LIN {X 0,Y 399.766,Z 653.208,A -85,B 0,C 180,E1 19416.646,E2 19416.646} C_VEL
LIN {X 0,Y 400.216,Z 637.351,A -85,B 0,C 180,E1 19415.617,E2 19415.617} C_VEL
LIN {X 0,Y 400.424,Z 621.306,A -85,B 0,C 180,E1 19414.872,E2 19414.872} C_VEL
LIN {X 0,Y 400.403,Z 603.741,A -85,B 0,C 180,E1 19414.34,E2 19414.34} C_VEL
LIN {X 0,Y 401.742,Z 547.411,A -85,B 0,C 180,E1 19413.015,E2 19413.015} C_VEL
LIN {X 0,Y 404.682,Z 475.698,A -85,B 0,C 180,E1 19411.198,E2 19411.198} C_VEL
LIN {X 0,Y 407.348,Z 462.24,A -85,B 0,C 180,E1 19410.277,E2 19410.277} C_VEL
LIN {X 0,Y 409.015,Z 418.407,A -85,B 0,C 180,E1 19406.548,E2 19406.548} C_VEL
LIN {X 0,Y 409.305,Z 412.468,A -85,B 0,C 180,E1 19406.028,E2 19406.028} C_VEL
LIN {X 0,Y 411.6,Z 412.53,A -85,B 0,C 180,E1 19405.697,E2 19405.697} C_VEL
LIN {X 0,Y 414.233,Z 411.427,A -85,B 0,C 180,E1 19405.443,E2 19405.443} C_VEL
LIN {X 0,Y 416.09,Z 410.465,A -85,B 0,C 180,E1 19405.285,E2 19405.285} C_VEL
LIN {X 0,Y 420.292,Z 409.112,A -85,B 0,C 180,E1 19404.851,E2 19404.851} C_VEL
LIN {X 0,Y 422.929,Z 408.049,A -85,B 0,C 180,E1 19404.605,E2 19404.605} C_VEL
LIN {X 0,Y 433.645,Z 404.285,A -85,B 0,C 180,E1 19403.595,E2 19403.595} C_VEL
LIN {X 0,Y 436.734,Z 421.547,A -85,B 0,C 180,E1 19401.653,E2 19401.653} C_VEL
LIN {X 0,Y 441.498,Z 436.637,A -85,B 0,C 180,E1 19399.802,E2 19399.802} C_VEL
LIN {X 0,Y 448.516,Z 451.234,A -85,B 0,C 180,E1 19397.856,E2 19397.856} C_VEL
LIN {X 0,Y 457.19,Z 463.962,A -85,B 0,C 180,E1 19396.015,E2 19396.015} C_VEL
LIN {X 0,Y 463.41,Z 471.327,A -85,B 0,C 180,E1 19394.895,E2 19394.895} C_VEL
LIN {X 0,Y 452.993,Z 490.31,A -85,B 0,C 180,E1 19394.314,E2 19394.314} C_VEL
LIN {X 0,Y 445.847,Z 504.974,A -85,B 0,C 180,E1 19393.771,E2 19393.771} C_VEL
LIN {X 0,Y 437.271,Z 522.126,A -85,B 0,C 180,E1 19393.133,E2 19393.133} C_VEL
LIN {X 0,Y 430.891,Z 538.04,A -85,B 0,C 180,E1 19392.428,E2 19392.428} C_VEL
LIN {X 0,Y 428.339,Z 556.287,A -85,B 0,C 180,E1 19392.311,E2 19392.311} C_VEL
LIN {X 0,Y 426.867,Z 574.916,A -85,B 0,C 180,E1 19392.06,E2 19392.06} C_VEL
LIN {X 0,Y 425.259,Z 601.251,A -85,B 0,C 180,E1 19391.436,E2 19391.436} C_VEL
LIN {X 0,Y 422.607,Z 628.36,A -85,B 0,C 180,E1 19390.562,E2 19390.562} C_VEL
LIN {X 0,Y 419.928,Z 652.409,A -85,B 0,C 180,E1 19389.516,E2 19389.516} C_VEL
LIN {X 0,Y 416.954,Z 675.906,A -85,B 0,C 180,E1 19388.221,E2 19388.221} C_VEL
LIN {X 0,Y 413.869,Z 698.687,A -85,B 0,C 180,E1 19386.672,E2 19386.672} C_VEL
LIN {X 0,Y 410.817,Z 719.469,A -85,B 0,C 180,E1 19384.972,E2 19384.972} C_VEL
LIN {X 0,Y 407.896,Z 738.189,A -85,B 0,C 180,E1 19383.136,E2 19383.136} C_VEL
LIN {X 0,Y 405.039,Z 755.282,A -85,B 0,C 180,E1 19381.142,E2 19381.142} C_VEL
LIN {X 0,Y 402.148,Z 771.736,A -85,B 0,C 180,E1 19378.839,E2 19378.839} C_VEL
LIN {X 0,Y 399.593,Z 786.158,A -85,B 0,C 180,E1 19376.448,E2 19376.448} C_VEL
LIN {X 0,Y 397.123,Z 800.578,A -85,B 0,C 180,E1 19373.587,E2 19373.587} C_VEL
LIN {X 0,Y 395.246,Z 812.426,A -85,B 0,C 180,E1 19370.742,E2 19370.742} C_VEL
LIN {X 0,Y 393.816,Z 822.794,A -85,B 0,C 180,E1 19367.738,E2 19367.738} C_VEL
LIN {X 0,Y 392.813,Z 832.018,A -85,B 0,C 180,E1 19364.445,E2 19364.445} C_VEL
LIN {X 0,Y 392.277,Z 839.142,A -85,B 0,C 180,E1 19361.17,E2 19361.17} C_VEL
LIN {X 0,Y 392.077,Z 843.984,A -85,B 0,C 180,E1 19358.21,E2 19358.21} C_VEL
LIN {X 0,Y 392.02,Z 847.572,A -85,B 0,C 180,E1 19354.975,E2 19354.975} C_VEL
LIN {X 0,Y 392.025,Z 849.318,A -85,B 0,C 180,E1 19351.9,E2 19351.9} C_VEL
LIN {X 0,Y 392.03,Z 849.521,A -85,B 0,C 180,E1 19348.831,E2 19348.831} C_VEL
LIN {X 0,Y 392.022,Z 848.087,A -85,B 0,C 180,E1 19345.745,E2 19345.745} C_VEL
LIN {X 0,Y 392.05,Z 845.113,A -85,B 0,C 180,E1 19342.674,E2 19342.674} C_VEL
LIN {X 0,Y 392.227,Z 840.178,A -85,B 0,C 180,E1 19339.424,E2 19339.424} C_VEL
LIN {X 0,Y 392.653,Z 833.716,A -85,B 0,C 180,E1 19336.301,E2 19336.301} C_VEL
LIN {X 0,Y 393.492,Z 825.441,A -85,B 0,C 180,E1 19333.161,E2 19333.161} C_VEL
LIN {X 0,Y 394.914,Z 814.562,A -85,B 0,C 180,E1 19329.859,E2 19329.859} C_VEL
LIN {X 0,Y 396.749,Z 802.631,A -85,B 0,C 180,E1 19326.903,E2 19326.903} C_VEL
LIN {X 0,Y 398.887,Z 790.123,A -85,B 0,C 180,E1 19324.301,E2 19324.301} C_VEL
LIN {X 0,Y 401.635,Z 774.648,A -85,B 0,C 180,E1 19321.609,E2 19321.609} C_VEL
LIN {X 0,Y 404.449,Z 758.875,A -85,B 0,C 180,E1 19319.311,E2 19319.311} C_VEL
LIN {X 0,Y 407.498,Z 741.326,A -85,B 0,C 180,E1 19317.162,E2 19317.162} C_VEL
LIN {X 0,Y 410.429,Z 723.021,A -85,B 0,C 180,E1 19315.307,E2 19315.307} C_VEL
LIN {X 0,Y 413.492,Z 703.01,A -85,B 0,C 180,E1 19313.584,E2 19313.584} C_VEL
LIN {X 0,Y 416.493,Z 681.937,A -85,B 0,C 180,E1 19312.079,E2 19312.079} C_VEL
LIN {X 0,Y 419.576,Z 658.834,A -85,B 0,C 180,E1 19310.711,E2 19310.711} C_VEL
LIN {X 0,Y 422.47,Z 635.021,A -85,B 0,C 180,E1 19309.591,E2 19309.591} C_VEL
LIN {X 0,Y 425.12,Z 610.015,A -85,B 0,C 180,E1 19308.697,E2 19308.697} C_VEL
LIN {X 0,Y 427.168,Z 584.161,A -85,B 0,C 180,E1 19308.01,E2 19308.01} C_VEL
LIN {X 0,Y 428.379,Z 565.366,A -85,B 0,C 180,E1 19307.66,E2 19307.66} C_VEL
LIN {X 0,Y 431.19,Z 543.77,A -85,B 0,C 180,E1 19307.511,E2 19307.511} C_VEL
LIN {X 0,Y 432.48,Z 537.146,A -85,B 0,C 180,E1 19307.494,E2 19307.494} C_VEL
LIN {X 0,Y 440.783,Z 520.892,A -85,B 0,C 180,E1 19306.671,E2 19306.671} C_VEL
LIN {X 0,Y 450.77,Z 504.788,A -85,B 0,C 180,E1 19306.03,E2 19306.03} C_VEL
LIN {X 0,Y 453.938,Z 499.823,A -85,B 0,C 180,E1 19305.846,E2 19305.846} C_VEL
LIN {X 0,Y 444.485,Z 487.571,A -85,B 0,C 180,E1 19303.855,E2 19303.855} C_VEL
LIN {X 0,Y 437.378,Z 474.491,A -85,B 0,C 180,E1 19301.875,E2 19301.875} C_VEL
LIN {X 0,Y 432.198,Z 460.151,A -85,B 0,C 180,E1 19299.852,E2 19299.852} C_VEL
LIN {X 0,Y 428.941,Z 443.777,A -85,B 0,C 180,E1 19297.725,E2 19297.725} C_VEL
LIN {X 0,Y 427.789,Z 425.876,A -85,B 0,C 180,E1 19295.589,E2 19295.589} C_VEL
LIN {X 0,Y 428.723,Z 407.137,A -85,B 0,C 180,E1 19293.554,E2 19293.554} C_VEL
LIN {X 0,Y 434.399,Z 369.568,A -85,B 0,C 180,E1 19289.85,E2 19289.85} C_VEL
LIN {X 0,Y 422.637,Z 374.64,A -85,B 0,C 180,E1 19288.547,E2 19288.547} C_VEL
LIN {X 0,Y 417.764,Z 376.744,A -85,B 0,C 180,E1 19287.975,E2 19287.975} C_VEL
LIN {X 0,Y 413.664,Z 378.626,A -85,B 0,C 180,E1 19287.494,E2 19287.494} C_VEL
LIN {X 0,Y 412.558,Z 378.969,A -85,B 0,C 180,E1 19287.339,E2 19287.339} C_VEL
LIN {X 0,Y 409.421,Z 380.815,A -85,B 0,C 180,E1 19287.015,E2 19287.015} C_VEL
LIN {X 0,Y 406.931,Z 381.358,A -85,B 0,C 180,E1 19286.581,E2 19286.581} C_VEL
LIN {X 0,Y 405.648,Z 427.519,A -85,B 0,C 180,E1 19282.996,E2 19282.996} C_VEL
LIN {X 0,Y 404.231,Z 473.732,A -85,B 0,C 180,E1 19279.356,E2 19279.356} C_VEL
LIN {X 0,Y 402.927,Z 508.519,A -85,B 0,C 180,E1 19276.581,E2 19276.581} C_VEL
LIN {X 0,Y 400.964,Z 520.121,A -85,B 0,C 180,E1 19275.813,E2 19275.813} C_VEL
LIN {X 0,Y 398.597,Z 615.75,A -85,B 0,C 180,E1 19273.629,E2 19273.629} C_VEL
LIN {X 0,Y 398.694,Z 635.16,A -85,B 0,C 180,E1 19273.118,E2 19273.118} C_VEL
LIN {X 0,Y 398.621,Z 649.308,A -85,B 0,C 180,E1 19272.494,E2 19272.494} C_VEL
LIN {X 0,Y 398.291,Z 663.605,A -85,B 0,C 180,E1 19271.585,E2 19271.585} C_VEL
LIN {X 0,Y 397.808,Z 676.96,A -85,B 0,C 180,E1 19270.426,E2 19270.426} C_VEL
LIN {X 0,Y 397.2,Z 689.029,A -85,B 0,C 180,E1 19269.051,E2 19269.051} C_VEL
LIN {X 0,Y 396.548,Z 699.323,A -85,B 0,C 180,E1 19267.533,E2 19267.533} C_VEL
LIN {X 0,Y 395.931,Z 707.723,A -85,B 0,C 180,E1 19265.942,E2 19265.942} C_VEL
LIN {X 0,Y 395.35,Z 714.813,A -85,B 0,C 180,E1 19264.205,E2 19264.205} C_VEL
LIN {X 0,Y 394.808,Z 720.81,A -85,B 0,C 180,E1 19262.177,E2 19262.177} C_VEL
LIN {X 0,Y 394.401,Z 724.738,A -85,B 0,C 180,E1 19260.145,E2 19260.145} C_VEL
LIN {X 0,Y 394.131,Z 726.813,A -85,B 0,C 180,E1 19258.11,E2 19258.11} C_VEL
LIN {X 0,Y 393.962,Z 727.145,A -85,B 0,C 180,E1 19256.07,E2 19256.07} C_VEL
LIN {X 0,Y 393.901,Z 725.545,A -85,B 0,C 180,E1 19253.879,E2 19253.879} C_VEL
LIN {X 0,Y 393.96,Z 721.902,A -85,B 0,C 180,E1 19251.682,E2 19251.682} C_VEL
LIN {X 0,Y 394.154,Z 716.495,A -85,B 0,C 180,E1 19249.623,E2 19249.623} C_VEL
LIN {X 0,Y 394.464,Z 709.492,A -85,B 0,C 180,E1 19247.706,E2 19247.706} C_VEL
LIN {X 0,Y 394.892,Z 701,A -85,B 0,C 180,E1 19245.932,E2 19245.932} C_VEL
LIN {X 0,Y 395.386,Z 691.035,A -85,B 0,C 180,E1 19244.3,E2 19244.3} C_VEL
LIN {X 0,Y 395.954,Z 678.81,A -85,B 0,C 180,E1 19242.739,E2 19242.739} C_VEL
LIN {X 0,Y 396.49,Z 665.133,A -85,B 0,C 180,E1 19241.397,E2 19241.397} C_VEL
LIN {X 0,Y 396.938,Z 650.985,A -85,B 0,C 180,E1 19240.349,E2 19240.349} C_VEL
LIN {X 0,Y 397.227,Z 635.067,A -85,B 0,C 180,E1 19239.51,E2 19239.51} C_VEL
LIN {X 0,Y 397.317,Z 618.736,A -85,B 0,C 180,E1 19238.972,E2 19238.972} C_VEL
LIN {X 0,Y 399.16,Z 507.374,A -85,B 0,C 180,E1 19236.646,E2 19236.646} C_VEL
LIN {X 0,Y 399.911,Z 499.645,A -85,B 0,C 180,E1 19236.028,E2 19236.028} C_VEL
LIN {X 0,Y 401.687,Z 449.496,A -85,B 0,C 180,E1 19231.855,E2 19231.855} C_VEL
LIN {X 0,Y 403.456,Z 402.025,A -85,B 0,C 180,E1 19227.887,E2 19227.887} C_VEL
LIN {X 0,Y 405.187,Z 356.102,A -85,B 0,C 180,E1 19224.034,E2 19224.034} C_VEL
LIN {X 0,Y 406.056,Z 332.68,A -85,B 0,C 180,E1 19222.049,E2 19222.049} C_VEL
LIN {X 0,Y 407.711,Z 332.474,A -85,B 0,C 180,E1 19221.65,E2 19221.65} C_VEL
LIN {X 0,Y 410.435,Z 330.957,A -85,B 0,C 180,E1 19221.238,E2 19221.238} C_VEL
LIN {X 0,Y 411.802,Z 330.204,A -85,B 0,C 180,E1 19221.034,E2 19221.034} C_VEL
LIN {X 0,Y 414.967,Z 328.853,A -85,B 0,C 180,E1 19220.497,E2 19220.497} C_VEL
LIN {X 0,Y 417.697,Z 327.456,A -85,B 0,C 180,E1 19220.094,E2 19220.094} C_VEL
LIN {X 0,Y 424.964,Z 324.13,A -85,B 0,C 180,E1 19218.993,E2 19218.993} C_VEL
LIN {X 0,Y 430.236,Z 337.107,A -85,B 0,C 180,E1 19215.708,E2 19215.708} C_VEL
LIN {X 0,Y 432.283,Z 343.09,A -85,B 0,C 180,E1 19214.38,E2 19214.38} C_VEL
LIN {X 0,Y 432.273,Z 344.872,A -85,B 0,C 180,E1 19214.218,E2 19214.218} C_VEL
LIN {X 0,Y 429.303,Z 421.475,A -85,B 0,C 180,E1 19212.78,E2 19212.78} C_VEL
LIN {X 0,Y 425.264,Z 492.221,A -85,B 0,C 180,E1 19211.237,E2 19211.237} C_VEL
LIN {X 0,Y 420.657,Z 559.279,A -85,B 0,C 180,E1 19209.571,E2 19209.571} C_VEL
LIN {X 0,Y 419.352,Z 566.901,A -85,B 0,C 180,E1 19209.458,E2 19209.458} C_VEL
LIN {X 0,Y 413.379,Z 586.126,A -85,B 0,C 180,E1 19209.411,E2 19209.411} C_VEL
LIN {X 0,Y 412.028,Z 593.598,A -85,B 0,C 180,E1 19209.224,E2 19209.224} C_VEL
LIN {X 0,Y 410.141,Z 613.958,A -85,B 0,C 180,E1 19208.31,E2 19208.31} C_VEL
LIN {X 0,Y 407.832,Z 633.355,A -85,B 0,C 180,E1 19207.175,E2 19207.175} C_VEL
LIN {X 0,Y 405.186,Z 652.171,A -85,B 0,C 180,E1 19205.792,E2 19205.792} C_VEL
LIN {X 0,Y 402.314,Z 670.111,A -85,B 0,C 180,E1 19204.172,E2 19204.172} C_VEL
LIN {X 0,Y 399.328,Z 687.129,A -85,B 0,C 180,E1 19202.315,E2 19202.315} C_VEL
LIN {X 0,Y 396.458,Z 702.616,A -85,B 0,C 180,E1 19200.292,E2 19200.292} C_VEL
LIN {X 0,Y 393.688,Z 717.186,A -85,B 0,C 180,E1 19198.025,E2 19198.025} C_VEL
LIN {X 0,Y 391.143,Z 730.612,A -85,B 0,C 180,E1 19195.529,E2 19195.529} C_VEL
LIN {X 0,Y 388.953,Z 742.643,A -85,B 0,C 180,E1 19192.841,E2 19192.841} C_VEL
LIN {X 0,Y 387.248,Z 752.834,A -85,B 0,C 180,E1 19190.084,E2 19190.084} C_VEL
LIN {X 0,Y 385.967,Z 761.558,A -85,B 0,C 180,E1 19187.177,E2 19187.177} C_VEL
LIN {X 0,Y 385.084,Z 768.742,A -85,B 0,C 180,E1 19184.127,E2 19184.127} C_VEL
LIN {X 0,Y 384.601,Z 774.069,A -85,B 0,C 180,E1 19181.092,E2 19181.092} C_VEL
LIN {X 0,Y 384.35,Z 777.624,A -85,B 0,C 180,E1 19178.076,E2 19178.076} C_VEL
LIN {X 0,Y 384.254,Z 779.455,A -85,B 0,C 180,E1 19175.225,E2 19175.225} C_VEL
LIN {X 0,Y 384.23,Z 779.823,A -85,B 0,C 180,E1 19172.186,E2 19172.186} C_VEL
LIN {X 0,Y 384.275,Z 778.608,A -85,B 0,C 180,E1 19169.255,E2 19169.255} C_VEL
LIN {X 0,Y 384.42,Z 775.983,A -85,B 0,C 180,E1 19166.421,E2 19166.421} C_VEL
LIN {X 0,Y 384.751,Z 771.574,A -85,B 0,C 180,E1 19163.434,E2 19163.434} C_VEL
LIN {X 0,Y 385.394,Z 765.21,A -85,B 0,C 180,E1 19160.359,E2 19160.359} C_VEL
LIN {X 0,Y 386.458,Z 756.918,A -85,B 0,C 180,E1 19157.296,E2 19157.296} C_VEL
LIN {X 0,Y 387.907,Z 747.238,A -85,B 0,C 180,E1 19154.451,E2 19154.451} C_VEL
LIN {X 0,Y 389.765,Z 736.08,A -85,B 0,C 180,E1 19151.762,E2 19151.762} C_VEL
LIN {X 0,Y 392.002,Z 723.467,A -85,B 0,C 180,E1 19149.235,E2 19149.235} C_VEL
LIN {X 0,Y 394.554,Z 709.375,A -85,B 0,C 180,E1 19146.871,E2 19146.871} C_VEL
LIN {X 0,Y 397.246,Z 694.286,A -85,B 0,C 180,E1 19144.746,E2 19144.746} C_VEL
LIN {X 0,Y 399.993,Z 678.33,A -85,B 0,C 180,E1 19142.861,E2 19142.861} C_VEL
LIN {X 0,Y 402.782,Z 660.794,A -85,B 0,C 180,E1 19141.13,E2 19141.13} C_VEL
LIN {X 0,Y 405.317,Z 643.236,A -85,B 0,C 180,E1 19139.702,E2 19139.702} C_VEL
LIN {X 0,Y 407.722,Z 623.961,A -85,B 0,C 180,E1 19138.428,E2 19138.428} C_VEL
LIN {X 0,Y 409.782,Z 603.646,A -85,B 0,C 180,E1 19137.379,E2 19137.379} C_VEL
LIN {X 0,Y 411.374,Z 583.008,A -85,B 0,C 180,E1 19136.592,E2 19136.592} C_VEL
LIN {X 0,Y 415.255,Z 526.804,A -85,B 0,C 180,E1 19135.073,E2 19135.073} C_VEL
LIN {X 0,Y 419.863,Z 454.196,A -85,B 0,C 180,E1 19133.357,E2 19133.357} C_VEL
LIN {X 0,Y 423.008,Z 388.842,A -85,B 0,C 180,E1 19132.029,E2 19132.029} C_VEL
LIN {X 0,Y 424.714,Z 343.474,A -85,B 0,C 180,E1 19131.185,E2 19131.185} C_VEL
LIN {X 0,Y 424.993,Z 342.278,A -85,B 0,C 180,E1 19131.085,E2 19131.085} C_VEL
LIN {X 0,Y 418.504,Z 327.03,A -85,B 0,C 180,E1 19127.99,E2 19127.99} C_VEL
LIN {X 0,Y 412.073,Z 312.861,A -85,B 0,C 180,E1 19124.722,E2 19124.722} C_VEL
LIN {X 0,Y 405.745,Z 300.174,A -85,B 0,C 180,E1 19121.333,E2 19121.333} C_VEL
LIN {X 0,Y 400.637,Z 290.686,A -85,B 0,C 180,E1 19118.404,E2 19118.404} C_VEL
LIN {X 0,Y 397.897,Z 285.744,A -85,B 0,C 180,E1 19116.716,E2 19116.716} C_VEL
LIN {X 0,Y 396.462,Z 283.778,A -85,B 0,C 180,E1 19115.899,E2 19115.899} C_VEL
LIN {X 0,Y 393.312,Z 284.578,A -85,B 0,C 180,E1 19115.057,E2 19115.057} C_VEL
LIN {X 0,Y 392.824,Z 284.611,A -85,B 0,C 180,E1 19114.828,E2 19114.828} C_VEL
LIN {X 0,Y 400.242,Z 307.24,A -85,B 0,C 180,E1 19112.064,E2 19112.064} C_VEL
LIN {X 0,Y 398.714,Z 347.658,A -85,B 0,C 180,E1 19108.384,E2 19108.384} C_VEL
LIN {X 0,Y 396.964,Z 390.836,A -85,B 0,C 180,E1 19104.478,E2 19104.478} C_VEL
LIN {X 0,Y 395.147,Z 435.751,A -85,B 0,C 180,E1 19100.438,E2 19100.438} C_VEL
LIN {X 0,Y 394.219,Z 458.804,A -85,B 0,C 180,E1 19098.408,E2 19098.408} C_VEL
LIN {X 0,Y 391.139,Z 602.019,A -85,B 0,C 180,E1 19095.262,E2 19095.262} C_VEL
LIN {X 0,Y 390.873,Z 620.072,A -85,B 0,C 180,E1 19094.594,E2 19094.594} C_VEL
LIN {X 0,Y 390.392,Z 636.284,A -85,B 0,C 180,E1 19093.705,E2 19093.705} C_VEL
LIN {X 0,Y 389.778,Z 651.493,A -85,B 0,C 180,E1 19092.595,E2 19092.595} C_VEL
LIN {X 0,Y 389.06,Z 666.417,A -85,B 0,C 180,E1 19091.189,E2 19091.189} C_VEL
LIN {X 0,Y 388.293,Z 679.992,A -85,B 0,C 180,E1 19089.561,E2 19089.561} C_VEL
LIN {X 0,Y 387.612,Z 691.431,A -85,B 0,C 180,E1 19087.858,E2 19087.858} C_VEL
LIN {X 0,Y 386.974,Z 702.533,A -85,B 0,C 180,E1 19085.784,E2 19085.784} C_VEL
LIN {X 0,Y 386.511,Z 711.159,A -85,B 0,C 180,E1 19083.709,E2 19083.709} C_VEL
LIN {X 0,Y 386.231,Z 717.878,A -85,B 0,C 180,E1 19081.632,E2 19081.632} C_VEL
LIN {X 0,Y 386.057,Z 723.403,A -85,B 0,C 180,E1 19079.259,E2 19079.259} C_VEL
LIN {X 0,Y 386.042,Z 726.72,A -85,B 0,C 180,E1 19077.031,E2 19077.031} C_VEL
LIN {X 0,Y 386.164,Z 728.422,A -85,B 0,C 180,E1 19074.652,E2 19074.652} C_VEL
LIN {X 0,Y 386.4,Z 728.138,A -85,B 0,C 180,E1 19072.337,E2 19072.337} C_VEL
LIN {X 0,Y 386.75,Z 726.237,A -85,B 0,C 180,E1 19070.176,E2 19070.176} C_VEL
LIN {X 0,Y 387.244,Z 722.377,A -85,B 0,C 180,E1 19067.928,E2 19067.928} C_VEL
LIN {X 0,Y 387.857,Z 716.957,A -85,B 0,C 180,E1 19065.825,E2 19065.825} C_VEL
LIN {X 0,Y 388.626,Z 709.429,A -85,B 0,C 180,E1 19063.714,E2 19063.714} C_VEL
LIN {X 0,Y 389.423,Z 701.004,A -85,B 0,C 180,E1 19061.901,E2 19061.901} C_VEL
LIN {X 0,Y 390.333,Z 690.067,A -85,B 0,C 180,E1 19060.068,E2 19060.068} C_VEL
LIN {X 0,Y 391.152,Z 678.727,A -85,B 0,C 180,E1 19058.56,E2 19058.56} C_VEL
LIN {X 0,Y 391.911,Z 665.72,A -85,B 0,C 180,E1 19057.184,E2 19057.184} C_VEL
LIN {X 0,Y 392.542,Z 650.586,A -85,B 0,C 180,E1 19055.95,E2 19055.95} C_VEL
LIN {X 0,Y 392.952,Z 635.394,A -85,B 0,C 180,E1 19055.015,E2 19055.015} C_VEL
LIN {X 0,Y 393.148,Z 619.173,A -85,B 0,C 180,E1 19054.303,E2 19054.303} C_VEL
LIN {X 0,Y 393.183,Z 593.979,A -85,B 0,C 180,E1 19053.616,E2 19053.616} C_VEL
LIN {X 0,Y 396.115,Z 513.758,A -85,B 0,C 180,E1 19051.594,E2 19051.594} C_VEL
LIN {X 0,Y 397.796,Z 478.237,A -85,B 0,C 180,E1 19050.651,E2 19050.651} C_VEL
LIN {X 0,Y 400.749,Z 464.037,A -85,B 0,C 180,E1 19049.685,E2 19049.685} C_VEL
LIN {X 0,Y 402.616,Z 421.711,A -85,B 0,C 180,E1 19046.03,E2 19046.03} C_VEL
LIN {X 0,Y 404.743,Z 421.756,A -85,B 0,C 180,E1 19045.72,E2 19045.72} C_VEL
LIN {X 0,Y 408.337,Z 420.092,A -85,B 0,C 180,E1 19045.384,E2 19045.384} C_VEL
LIN {X 0,Y 413.437,Z 418.339,A -85,B 0,C 180,E1 19044.86,E2 19044.86} C_VEL
LIN {X 0,Y 416.139,Z 417.134,A -85,B 0,C 180,E1 19044.617,E2 19044.617} C_VEL
LIN {X 0,Y 427.999,Z 412.848,A -85,B 0,C 180,E1 19043.498,E2 19043.498} C_VEL
LIN {X 0,Y 431.631,Z 430.284,A -85,B 0,C 180,E1 19041.455,E2 19041.455} C_VEL
LIN {X 0,Y 437.129,Z 445.653,A -85,B 0,C 180,E1 19039.489,E2 19039.489} C_VEL
LIN {X 0,Y 444.538,Z 459.767,A -85,B 0,C 180,E1 19037.54,E2 19037.54} C_VEL
LIN {X 0,Y 454.237,Z 472.872,A -85,B 0,C 180,E1 19035.575,E2 19035.575} C_VEL
LIN {X 0,Y 454.987,Z 473.978,A -85,B 0,C 180,E1 19035.422,E2 19035.422} C_VEL
LIN {X 0,Y 444.847,Z 493.092,A -85,B 0,C 180,E1 19034.801,E2 19034.801} C_VEL
LIN {X 0,Y 439.941,Z 503.129,A -85,B 0,C 180,E1 19034.427,E2 19034.427} C_VEL
LIN {X 0,Y 430.848,Z 521.237,A -85,B 0,C 180,E1 19033.754,E2 19033.754} C_VEL
LIN {X 0,Y 424.984,Z 535.777,A -85,B 0,C 180,E1 19033.115,E2 19033.115} C_VEL
LIN {X 0,Y 422.179,Z 555.484,A -85,B 0,C 180,E1 19032.995,E2 19032.995} C_VEL
LIN {X 0,Y 420.575,Z 575.072,A -85,B 0,C 180,E1 19032.729,E2 19032.729} C_VEL
LIN {X 0,Y 418.677,Z 602.883,A -85,B 0,C 180,E1 19032.037,E2 19032.037} C_VEL
LIN {X 0,Y 415.982,Z 628.895,A -85,B 0,C 180,E1 19031.17,E2 19031.17} C_VEL
LIN {X 0,Y 413.011,Z 653.938,A -85,B 0,C 180,E1 19030.043,E2 19030.043} C_VEL
LIN {X 0,Y 409.821,Z 678.02,A -85,B 0,C 180,E1 19028.674,E2 19028.674} C_VEL
LIN {X 0,Y 406.671,Z 700.048,A -85,B 0,C 180,E1 19027.128,E2 19027.128} C_VEL
LIN {X 0,Y 403.469,Z 720.766,A -85,B 0,C 180,E1 19025.382,E2 19025.382} C_VEL
LIN {X 0,Y 400.396,Z 739.668,A -85,B 0,C 180,E1 19023.483,E2 19023.483} C_VEL
LIN {X 0,Y 397.465,Z 756.218,A -85,B 0,C 180,E1 19021.485,E2 19021.485} C_VEL
LIN {X 0,Y 394.453,Z 772.679,A -85,B 0,C 180,E1 19019.123,E2 19019.123} C_VEL
LIN {X 0,Y 391.654,Z 787.691,A -85,B 0,C 180,E1 19016.536,E2 19016.536} C_VEL
LIN {X 0,Y 389.349,Z 800.535,A -85,B 0,C 180,E1 19013.906,E2 19013.906} C_VEL
LIN {X 0,Y 387.293,Z 812.986,A -85,B 0,C 180,E1 19010.844,E2 19010.844} C_VEL
LIN {X 0,Y 385.834,Z 823.088,A -85,B 0,C 180,E1 19007.806,E2 19007.806} C_VEL
LIN {X 0,Y 384.877,Z 831.385,A -85,B 0,C 180,E1 19004.749,E2 19004.749} C_VEL
LIN {X 0,Y 384.305,Z 838.495,A -85,B 0,C 180,E1 19001.404,E2 19001.404} C_VEL
LIN {X 0,Y 384.091,Z 843.498,A -85,B 0,C 180,E1 18998.232,E2 18998.232} C_VEL
LIN {X 0,Y 384.043,Z 846.875,A -85,B 0,C 180,E1 18995.078,E2 18995.078} C_VEL
LIN {X 0,Y 384.056,Z 848.606,A -85,B 0,C 180,E1 18991.939,E2 18991.939} C_VEL
LIN {X 0,Y 384.061,Z 848.805,A -85,B 0,C 180,E1 18988.807,E2 18988.807} C_VEL
LIN {X 0,Y 384.048,Z 847.375,A -85,B 0,C 180,E1 18985.652,E2 18985.652} C_VEL
LIN {X 0,Y 384.066,Z 844.421,A -85,B 0,C 180,E1 18982.521,E2 18982.521} C_VEL
LIN {X 0,Y 384.251,Z 839.501,A -85,B 0,C 180,E1 18979.202,E2 18979.202} C_VEL
LIN {X 0,Y 384.708,Z 833.07,A -85,B 0,C 180,E1 18976.012,E2 18976.012} C_VEL
LIN {X 0,Y 385.607,Z 824.804,A -85,B 0,C 180,E1 18972.807,E2 18972.807} C_VEL
LIN {X 0,Y 386.988,Z 814.814,A -85,B 0,C 180,E1 18969.697,E2 18969.697} C_VEL
LIN {X 0,Y 388.79,Z 803.699,A -85,B 0,C 180,E1 18966.829,E2 18966.829} C_VEL
LIN {X 0,Y 391.221,Z 790.127,A -85,B 0,C 180,E1 18963.922,E2 18963.922} C_VEL
LIN {X 0,Y 393.931,Z 775.664,A -85,B 0,C 180,E1 18961.333,E2 18961.333} C_VEL
LIN {X 0,Y 396.975,Z 759.557,A -85,B 0,C 180,E1 18958.909,E2 18958.909} C_VEL
LIN {X 0,Y 400.135,Z 742.218,A -85,B 0,C 180,E1 18956.736,E2 18956.736} C_VEL
LIN {X 0,Y 403.172,Z 724.463,A -85,B 0,C 180,E1 18954.875,E2 18954.875} C_VEL
LIN {X 0,Y 406.397,Z 704.128,A -85,B 0,C 180,E1 18953.091,E2 18953.091} C_VEL
LIN {X 0,Y 409.744,Z 681.859,A -85,B 0,C 180,E1 18951.463,E2 18951.463} C_VEL
LIN {X 0,Y 412.856,Z 659.708,A -85,B 0,C 180,E1 18950.125,E2 18950.125} C_VEL
LIN {X 0,Y 415.898,Z 635.987,A -85,B 0,C 180,E1 18948.98,E2 18948.98} C_VEL
LIN {X 0,Y 418.706,Z 611.267,A -85,B 0,C 180,E1 18948.061,E2 18948.061} C_VEL
LIN {X 0,Y 421.024,Z 583.9,A -85,B 0,C 180,E1 18947.311,E2 18947.311} C_VEL
LIN {X 0,Y 422.297,Z 565.542,A -85,B 0,C 180,E1 18946.959,E2 18946.959} C_VEL
LIN {X 0,Y 425.177,Z 543.452,A -85,B 0,C 180,E1 18946.802,E2 18946.802} C_VEL
LIN {X 0,Y 426.751,Z 534.834,A -85,B 0,C 180,E1 18946.785,E2 18946.785} C_VEL
LIN {X 0,Y 435.293,Z 518.473,A -85,B 0,C 180,E1 18945.968,E2 18945.968} C_VEL
LIN {X 0,Y 445.416,Z 502.173,A -85,B 0,C 180,E1 18945.323,E2 18945.323} C_VEL
LIN {X 0,Y 436.31,Z 489.424,A -85,B 0,C 180,E1 18943.25,E2 18943.25} C_VEL
LIN {X 0,Y 429.248,Z 474.91,A -85,B 0,C 180,E1 18941.061,E2 18941.061} C_VEL
LIN {X 0,Y 424.621,Z 459.897,A -85,B 0,C 180,E1 18938.954,E2 18938.954} C_VEL
LIN {X 0,Y 422.013,Z 443.175,A -85,B 0,C 180,E1 18936.792,E2 18936.792} C_VEL
LIN {X 0,Y 421.482,Z 424.669,A -85,B 0,C 180,E1 18934.596,E2 18934.596} C_VEL
LIN {X 0,Y 423.154,Z 404.59,A -85,B 0,C 180,E1 18932.437,E2 18932.437} C_VEL
LIN {X 0,Y 427.236,Z 378.504,A -85,B 0,C 180,E1 18929.822,E2 18929.822} C_VEL
LIN {X 0,Y 416.005,Z 383.444,A -85,B 0,C 180,E1 18928.573,E2 18928.573} C_VEL
LIN {X 0,Y 411.032,Z 385.656,A -85,B 0,C 180,E1 18927.99,E2 18927.99} C_VEL
LIN {X 0,Y 406.926,Z 387.609,A -85,B 0,C 180,E1 18927.512,E2 18927.512} C_VEL
LIN {X 0,Y 405.329,Z 388.293,A -85,B 0,C 180,E1 18927.311,E2 18927.311} C_VEL
LIN {X 0,Y 401.868,Z 390.174,A -85,B 0,C 180,E1 18926.924,E2 18926.924} C_VEL
LIN {X 0,Y 399.988,Z 390.421,A -85,B 0,C 180,E1 18926.58,E2 18926.58} C_VEL
LIN {X 0,Y 398.658,Z 433.584,A -85,B 0,C 180,E1 18923.188,E2 18923.188} C_VEL
LIN {X 0,Y 396.964,Z 481.671,A -85,B 0,C 180,E1 18919.342,E2 18919.342} C_VEL
LIN {X 0,Y 395.872,Z 509.249,A -85,B 0,C 180,E1 18917.112,E2 18917.112} C_VEL
LIN {X 0,Y 393.709,Z 521.923,A -85,B 0,C 180,E1 18916.276,E2 18916.276} C_VEL
LIN {X 0,Y 391.15,Z 614.357,A -85,B 0,C 180,E1 18914.087,E2 18914.087} C_VEL
LIN {X 0,Y 391.211,Z 636.405,A -85,B 0,C 180,E1 18913.495,E2 18913.495} C_VEL
LIN {X 0,Y 391.121,Z 650.744,A -85,B 0,C 180,E1 18912.85,E2 18912.85} C_VEL
LIN {X 0,Y 390.786,Z 664.603,A -85,B 0,C 180,E1 18911.96,E2 18911.96} C_VEL
LIN {X 0,Y 390.273,Z 678.119,A -85,B 0,C 180,E1 18910.779,E2 18910.779} C_VEL
LIN {X 0,Y 389.615,Z 690.255,A -85,B 0,C 180,E1 18909.378,E2 18909.378} C_VEL
LIN {X 0,Y 388.908,Z 700.587,A -85,B 0,C 180,E1 18907.831,E2 18907.831} C_VEL
LIN {X 0,Y 388.243,Z 709.042,A -85,B 0,C 180,E1 18906.209,E2 18906.209} C_VEL
LIN {X 0,Y 387.615,Z 716.181,A -85,B 0,C 180,E1 18904.438,E2 18904.438} C_VEL
LIN {X 0,Y 387.023,Z 722.204,A -85,B 0,C 180,E1 18902.368,E2 18902.368} C_VEL
LIN {X 0,Y 386.574,Z 726.129,A -85,B 0,C 180,E1 18900.296,E2 18900.296} C_VEL
LIN {X 0,Y 386.27,Z 728.194,A -85,B 0,C 180,E1 18898.219,E2 18898.219} C_VEL
LIN {X 0,Y 386.082,Z 728.516,A -85,B 0,C 180,E1 18896.139,E2 18896.139} C_VEL
LIN {X 0,Y 386.007,Z 726.886,A -85,B 0,C 180,E1 18893.903,E2 18893.903} C_VEL
LIN {X 0,Y 386.061,Z 723.199,A -85,B 0,C 180,E1 18891.66,E2 18891.66} C_VEL
LIN {X 0,Y 386.259,Z 717.737,A -85,B 0,C 180,E1 18889.56,E2 18889.56} C_VEL
LIN {X 0,Y 386.579,Z 710.673,A -85,B 0,C 180,E1 18887.603,E2 18887.603} C_VEL
LIN {X 0,Y 387.023,Z 702.099,A -85,B 0,C 180,E1 18885.792,E2 18885.792} C_VEL
LIN {X 0,Y 387.536,Z 692.041,A -85,B 0,C 180,E1 18884.128,E2 18884.128} C_VEL
LIN {X 0,Y 388.098,Z 680.383,A -85,B 0,C 180,E1 18882.611,E2 18882.611} C_VEL
LIN {X 0,Y 388.654,Z 666.785,A -85,B 0,C 180,E1 18881.241,E2 18881.241} C_VEL
LIN {X 0,Y 389.142,Z 651.95,A -85,B 0,C 180,E1 18880.12,E2 18880.12} C_VEL
LIN {X 0,Y 389.44,Z 636.116,A -85,B 0,C 180,E1 18879.272,E2 18879.272} C_VEL
LIN {X 0,Y 389.537,Z 620.018,A -85,B 0,C 180,E1 18878.728,E2 18878.728} C_VEL
LIN {X 0,Y 391.501,Z 508.362,A -85,B 0,C 180,E1 18876.321,E2 18876.321} C_VEL
LIN {X 0,Y 392.306,Z 500.461,A -85,B 0,C 180,E1 18875.687,E2 18875.687} C_VEL
LIN {X 0,Y 394.144,Z 450.74,A -85,B 0,C 180,E1 18871.515,E2 18871.515} C_VEL
LIN {X 0,Y 395.974,Z 403.652,A -85,B 0,C 180,E1 18867.548,E2 18867.548} C_VEL
LIN {X 0,Y 397.784,Z 358.292,A -85,B 0,C 180,E1 18863.704,E2 18863.704} C_VEL
LIN {X 0,Y 398.447,Z 341.738,A -85,B 0,C 180,E1 18862.289,E2 18862.289} C_VEL
LIN {X 0,Y 400.097,Z 341.514,A -85,B 0,C 180,E1 18861.883,E2 18861.883} C_VEL
LIN {X 0,Y 402.817,Z 339.976,A -85,B 0,C 180,E1 18861.462,E2 18861.462} C_VEL
LIN {X 0,Y 404.207,Z 339.161,A -85,B 0,C 180,E1 18861.256,E2 18861.256} C_VEL
LIN {X 0,Y 407.373,Z 337.768,A -85,B 0,C 180,E1 18860.71,E2 18860.71} C_VEL
LIN {X 0,Y 409.491,Z 336.54,A -85,B 0,C 180,E1 18860.409,E2 18860.409} C_VEL
LIN {X 0,Y 414.15,Z 334.337,A -85,B 0,C 180,E1 18859.682,E2 18859.682} C_VEL
LIN {X 0,Y 420.222,Z 331.519,A -85,B 0,C 180,E1 18858.769,E2 18858.769} C_VEL
LIN {X 0,Y 424.852,Z 343.012,A -85,B 0,C 180,E1 18855.843,E2 18855.843} C_VEL
LIN {X 0,Y 426.425,Z 346.976,A -85,B 0,C 180,E1 18854.965,E2 18854.965} C_VEL
LIN {X 0,Y 423.791,Z 417.102,A -85,B 0,C 180,E1 18853.621,E2 18853.621} C_VEL
LIN {X 0,Y 419.867,Z 484.325,A -85,B 0,C 180,E1 18852.158,E2 18852.158} C_VEL
LIN {X 0,Y 414.387,Z 560.55,A -85,B 0,C 180,E1 18850.239,E2 18850.239} C_VEL
LIN {X 0,Y 412.259,Z 590.931,A -85,B 0,C 180,E1 18849.327,E2 18849.327} C_VEL
LIN {X 0,Y 412.028,Z 593.598,A -85,B 0,C 180,E1 18849.224,E2 18849.224} C_VEL
LIN {X 0,Y 410.598,Z 601.182,A -85,B 0,C 180,E1 18849.009,E2 18849.009} C_VEL
LIN {X 0,Y 403.936,Z 619.978,A -85,B 0,C 180,E1 18848.614,E2 18848.614} C_VEL
LIN {X 0,Y 402.285,Z 627.038,A -85,B 0,C 180,E1 18848.286,E2 18848.286} C_VEL
LIN {X 0,Y 399.658,Z 645.895,A -85,B 0,C 180,E1 18846.991,E2 18846.991} C_VEL
LIN {X 0,Y 396.685,Z 664.294,A -85,B 0,C 180,E1 18845.432,E2 18845.432} C_VEL
LIN {X 0,Y 393.585,Z 681.711,A -85,B 0,C 180,E1 18843.629,E2 18843.629} C_VEL
LIN {X 0,Y 390.416,Z 698.127,A -85,B 0,C 180,E1 18841.587,E2 18841.587} C_VEL
LIN {X 0,Y 387.43,Z 713.045,A -85,B 0,C 180,E1 18839.363,E2 18839.363} C_VEL
LIN {X 0,Y 384.617,Z 726.919,A -85,B 0,C 180,E1 18836.894,E2 18836.894} C_VEL
LIN {X 0,Y 382.169,Z 739.298,A -85,B 0,C 180,E1 18834.253,E2 18834.253} C_VEL
LIN {X 0,Y 380.098,Z 750.437,A -85,B 0,C 180,E1 18831.374,E2 18831.374} C_VEL
LIN {X 0,Y 378.512,Z 760,A -85,B 0,C 180,E1 18828.321,E2 18828.321} C_VEL
LIN {X 0,Y 377.415,Z 767.702,A -85,B 0,C 180,E1 18825.205,E2 18825.205} C_VEL
LIN {X 0,Y 376.78,Z 773.497,A -85,B 0,C 180,E1 18822.102,E2 18822.102} C_VEL
LIN {X 0,Y 376.453,Z 777.53,A -85,B 0,C 180,E1 18819.016,E2 18819.016} C_VEL
LIN {X 0,Y 376.312,Z 779.83,A -85,B 0,C 180,E1 18816.101,E2 18816.101} C_VEL
LIN {X 0,Y 376.268,Z 780.658,A -85,B 0,C 180,E1 18813.047,E2 18813.047} C_VEL
LIN {X 0,Y 376.301,Z 779.822,A -85,B 0,C 180,E1 18810,E2 18810} C_VEL
LIN {X 0,Y 376.406,Z 777.541,A -85,B 0,C 180,E1 18807.107,E2 18807.107} C_VEL
LIN {X 0,Y 376.71,Z 773.563,A -85,B 0,C 180,E1 18804.059,E2 18804.059} C_VEL
LIN {X 0,Y 377.282,Z 767.875,A -85,B 0,C 180,E1 18801.004,E2 18801.004} C_VEL
LIN {X 0,Y 378.25,Z 760.429,A -85,B 0,C 180,E1 18797.976,E2 18797.976} C_VEL
LIN {X 0,Y 379.582,Z 751.806,A -85,B 0,C 180,E1 18795.179,E2 18795.179} C_VEL
LIN {X 0,Y 381.355,Z 741.547,A -85,B 0,C 180,E1 18792.451,E2 18792.451} C_VEL
LIN {X 0,Y 383.603,Z 729.385,A -85,B 0,C 180,E1 18789.776,E2 18789.776} C_VEL
LIN {X 0,Y 386.176,Z 715.927,A -85,B 0,C 180,E1 18787.308,E2 18787.308} C_VEL
LIN {X 0,Y 389.058,Z 700.812,A -85,B 0,C 180,E1 18784.991,E2 18784.991} C_VEL
LIN {X 0,Y 392.037,Z 684.629,A -85,B 0,C 180,E1 18782.919,E2 18782.919} C_VEL
LIN {X 0,Y 395,Z 667.438,A -85,B 0,C 180,E1 18781.087,E2 18781.087} C_VEL
LIN {X 0,Y 397.844,Z 649.277,A -85,B 0,C 180,E1 18779.491,E2 18779.491} C_VEL
LIN {X 0,Y 400.473,Z 630.099,A -85,B 0,C 180,E1 18778.126,E2 18778.126} C_VEL
LIN {X 0,Y 402.69,Z 610.383,A -85,B 0,C 180,E1 18777.014,E2 18777.014} C_VEL
LIN {X 0,Y 404.52,Z 589.455,A -85,B 0,C 180,E1 18776.128,E2 18776.128} C_VEL
LIN {X 0,Y 407.393,Z 549.034,A -85,B 0,C 180,E1 18774.949,E2 18774.949} C_VEL
LIN {X 0,Y 412.523,Z 476.301,A -85,B 0,C 180,E1 18773.125,E2 18773.125} C_VEL
LIN {X 0,Y 416.208,Z 410.878,A -85,B 0,C 180,E1 18771.712,E2 18771.712} C_VEL
LIN {X 0,Y 418.719,Z 345.943,A -85,B 0,C 180,E1 18770.471,E2 18770.471} C_VEL
LIN {X 0,Y 412.3,Z 330.667,A -85,B 0,C 180,E1 18767.291,E2 18767.291} C_VEL
LIN {X 0,Y 406.26,Z 317.516,A -85,B 0,C 180,E1 18764.148,E2 18764.148} C_VEL
LIN {X 0,Y 400.656,Z 306.026,A -85,B 0,C 180,E1 18761.021,E2 18761.021} C_VEL
LIN {X 0,Y 395.666,Z 296.654,A -85,B 0,C 180,E1 18758.069,E2 18758.069} C_VEL
LIN {X 0,Y 392.974,Z 291.781,A -85,B 0,C 180,E1 18756.359,E2 18756.359} C_VEL
LIN {X 0,Y 392.302,Z 290.909,A -85,B 0,C 180,E1 18755.979,E2 18755.979} C_VEL
LIN {X 0,Y 387.678,Z 292.281,A -85,B 0,C 180,E1 18754.75,E2 18754.75} C_VEL
LIN {X 0,Y 387.291,Z 292.283,A -85,B 0,C 180,E1 18754.557,E2 18754.557} C_VEL
LIN {X 0,Y 392.947,Z 309.789,A -85,B 0,C 180,E1 18752.41,E2 18752.41} C_VEL
LIN {X 0,Y 391.31,Z 350.965,A -85,B 0,C 180,E1 18748.627,E2 18748.627} C_VEL
LIN {X 0,Y 389.481,Z 393.623,A -85,B 0,C 180,E1 18744.737,E2 18744.737} C_VEL
LIN {X 0,Y 387.589,Z 438.123,A -85,B 0,C 180,E1 18740.697,E2 18740.697} C_VEL
LIN {X 0,Y 386.648,Z 459.829,A -85,B 0,C 180,E1 18738.777,E2 18738.777} C_VEL
LIN {X 0,Y 383.396,Z 602.42,A -85,B 0,C 180,E1 18735.553,E2 18735.553} C_VEL
LIN {X 0,Y 383.123,Z 620.344,A -85,B 0,C 180,E1 18734.887,E2 18734.887} C_VEL
LIN {X 0,Y 382.648,Z 636.334,A -85,B 0,C 180,E1 18734.012,E2 18734.012} C_VEL
LIN {X 0,Y 382.001,Z 652.152,A -85,B 0,C 180,E1 18732.855,E2 18732.855} C_VEL
LIN {X 0,Y 381.254,Z 667.215,A -85,B 0,C 180,E1 18731.421,E2 18731.421} C_VEL
LIN {X 0,Y 380.494,Z 680.372,A -85,B 0,C 180,E1 18729.835,E2 18729.835} C_VEL
LIN {X 0,Y 379.815,Z 691.604,A -85,B 0,C 180,E1 18728.173,E2 18728.173} C_VEL
LIN {X 0,Y 379.171,Z 702.237,A -85,B 0,C 180,E1 18726.205,E2 18726.205} C_VEL
LIN {X 0,Y 378.713,Z 710.755,A -85,B 0,C 180,E1 18724.24,E2 18724.24} C_VEL
LIN {X 0,Y 378.362,Z 718.328,A -85,B 0,C 180,E1 18721.969,E2 18721.969} C_VEL
LIN {X 0,Y 378.191,Z 723.586,A -85,B 0,C 180,E1 18719.849,E2 18719.849} C_VEL
LIN {X 0,Y 378.146,Z 727.621,A -85,B 0,C 180,E1 18717.424,E2 18717.424} C_VEL
LIN {X 0,Y 378.251,Z 729.602,A -85,B 0,C 180,E1 18715.148,E2 18715.148} C_VEL
LIN {X 0,Y 378.473,Z 729.889,A -85,B 0,C 180,E1 18712.868,E2 18712.868} C_VEL
LIN {X 0,Y 378.832,Z 728.381,A -85,B 0,C 180,E1 18710.582,E2 18710.582} C_VEL
LIN {X 0,Y 379.352,Z 725.067,A -85,B 0,C 180,E1 18708.291,E2 18708.291} C_VEL
LIN {X 0,Y 379.968,Z 720.135,A -85,B 0,C 180,E1 18706.146,E2 18706.146} C_VEL
LIN {X 0,Y 380.776,Z 713.229,A -85,B 0,C 180,E1 18703.996,E2 18703.996} C_VEL
LIN {X 0,Y 381.674,Z 704.546,A -85,B 0,C 180,E1 18701.98,E2 18701.98} C_VEL
LIN {X 0,Y 382.607,Z 694.674,A -85,B 0,C 180,E1 18700.184,E2 18700.184} C_VEL
LIN {X 0,Y 383.519,Z 683.252,A -85,B 0,C 180,E1 18698.549,E2 18698.549} C_VEL
LIN {X 0,Y 384.358,Z 670.567,A -85,B 0,C 180,E1 18697.106,E2 18697.106} C_VEL
LIN {X 0,Y 385.063,Z 656.69,A -85,B 0,C 180,E1 18695.861,E2 18695.861} C_VEL
LIN {X 0,Y 385.612,Z 640.237,A -85,B 0,C 180,E1 18694.753,E2 18694.753} C_VEL
LIN {X 0,Y 385.905,Z 622.714,A -85,B 0,C 180,E1 18693.914,E2 18693.914} C_VEL
LIN {X 0,Y 385.927,Z 601.494,A -85,B 0,C 180,E1 18693.28,E2 18693.28} C_VEL
LIN {X 0,Y 388.394,Z 533.469,A -85,B 0,C 180,E1 18691.507,E2 18691.507} C_VEL
LIN {X 0,Y 391.198,Z 480.146,A -85,B 0,C 180,E1 18690.022,E2 18690.022} C_VEL
LIN {X 0,Y 394.301,Z 465.434,A -85,B 0,C 180,E1 18689.019,E2 18689.019} C_VEL
LIN {X 0,Y 396.053,Z 431.065,A -85,B 0,C 180,E1 18686.001,E2 18686.001} C_VEL
LIN {X 0,Y 398.625,Z 430.916,A -85,B 0,C 180,E1 18685.643,E2 18685.643} C_VEL
LIN {X 0,Y 402.593,Z 428.855,A -85,B 0,C 180,E1 18685.292,E2 18685.292} C_VEL
LIN {X 0,Y 406.568,Z 427.588,A -85,B 0,C 180,E1 18684.868,E2 18684.868} C_VEL
LIN {X 0,Y 409.284,Z 426.351,A -85,B 0,C 180,E1 18684.622,E2 18684.622} C_VEL
LIN {X 0,Y 422.454,Z 421.385,A -85,B 0,C 180,E1 18683.386,E2 18683.386} C_VEL
LIN {X 0,Y 426.469,Z 438.289,A -85,B 0,C 180,E1 18681.327,E2 18681.327} C_VEL
LIN {X 0,Y 432.246,Z 453.221,A -85,B 0,C 180,E1 18679.352,E2 18679.352} C_VEL
LIN {X 0,Y 439.973,Z 467.132,A -85,B 0,C 180,E1 18677.374,E2 18677.374} C_VEL
LIN {X 0,Y 446.715,Z 476.578,A -85,B 0,C 180,E1 18675.96,E2 18675.96} C_VEL
LIN {X 0,Y 437.238,Z 494.969,A -85,B 0,C 180,E1 18675.332,E2 18675.332} C_VEL
LIN {X 0,Y 432.125,Z 504.9,A -85,B 0,C 180,E1 18674.981,E2 18674.981} C_VEL
LIN {X 0,Y 423.235,Z 523.107,A -85,B 0,C 180,E1 18674.275,E2 18674.275} C_VEL
LIN {X 0,Y 419.112,Z 533.475,A -85,B 0,C 180,E1 18673.824,E2 18673.824} C_VEL
LIN {X 0,Y 416.022,Z 555.271,A -85,B 0,C 180,E1 18673.693,E2 18673.693} C_VEL
LIN {X 0,Y 414.313,Z 575.059,A -85,B 0,C 180,E1 18673.415,E2 18673.415} C_VEL
LIN {X 0,Y 412.212,Z 603.769,A -85,B 0,C 180,E1 18672.679,E2 18672.679} C_VEL
LIN {X 0,Y 409.377,Z 629.374,A -85,B 0,C 180,E1 18671.793,E2 18671.793} C_VEL
LIN {X 0,Y 406.304,Z 654.143,A -85,B 0,C 180,E1 18670.656,E2 18670.656} C_VEL
LIN {X 0,Y 403.003,Z 677.964,A -85,B 0,C 180,E1 18669.279,E2 18669.279} C_VEL
LIN {X 0,Y 399.556,Z 700.936,A -85,B 0,C 180,E1 18667.633,E2 18667.633} C_VEL
LIN {X 0,Y 396.196,Z 721.773,A -85,B 0,C 180,E1 18665.838,E2 18665.838} C_VEL
LIN {X 0,Y 393.175,Z 739.514,A -85,B 0,C 180,E1 18664.019,E2 18664.019} C_VEL
LIN {X 0,Y 389.849,Z 757.443,A -85,B 0,C 180,E1 18661.802,E2 18661.802} C_VEL
LIN {X 0,Y 386.847,Z 772.996,A -85,B 0,C 180,E1 18659.497,E2 18659.497} C_VEL
LIN {X 0,Y 384.012,Z 787.554,A -85,B 0,C 180,E1 18656.94,E2 18656.94} C_VEL
LIN {X 0,Y 381.58,Z 800.428,A -85,B 0,C 180,E1 18654.236,E2 18654.236} C_VEL
LIN {X 0,Y 379.549,Z 812.105,A -85,B 0,C 180,E1 18651.318,E2 18651.318} C_VEL
LIN {X 0,Y 377.975,Z 822.367,A -85,B 0,C 180,E1 18648.189,E2 18648.189} C_VEL
LIN {X 0,Y 376.949,Z 830.702,A -85,B 0,C 180,E1 18645.067,E2 18645.067} C_VEL
LIN {X 0,Y 376.338,Z 837.837,A -85,B 0,C 180,E1 18641.649,E2 18641.649} C_VEL
LIN {X 0,Y 376.107,Z 842.817,A -85,B 0,C 180,E1 18638.408,E2 18638.408} C_VEL
LIN {X 0,Y 376.066,Z 846.18,A -85,B 0,C 180,E1 18635.186,E2 18635.186} C_VEL
LIN {X 0,Y 376.087,Z 847.893,A -85,B 0,C 180,E1 18631.981,E2 18631.981} C_VEL
LIN {X 0,Y 376.092,Z 848.088,A -85,B 0,C 180,E1 18628.781,E2 18628.781} C_VEL
LIN {X 0,Y 376.073,Z 846.678,A -85,B 0,C 180,E1 18625.578,E2 18625.578} C_VEL
LIN {X 0,Y 376.085,Z 843.724,A -85,B 0,C 180,E1 18622.361,E2 18622.361} C_VEL
LIN {X 0,Y 376.263,Z 839.084,A -85,B 0,C 180,E1 18619.125,E2 18619.125} C_VEL
LIN {X 0,Y 376.734,Z 832.768,A -85,B 0,C 180,E1 18615.867,E2 18615.867} C_VEL
LIN {X 0,Y 377.728,Z 824.115,A -85,B 0,C 180,E1 18612.436,E2 18612.436} C_VEL
LIN {X 0,Y 379.185,Z 814.27,A -85,B 0,C 180,E1 18609.308,E2 18609.308} C_VEL
LIN {X 0,Y 381.191,Z 802.664,A -85,B 0,C 180,E1 18606.265,E2 18606.265} C_VEL
LIN {X 0,Y 383.757,Z 789.146,A -85,B 0,C 180,E1 18603.337,E2 18603.337} C_VEL
LIN {X 0,Y 386.604,Z 774.81,A -85,B 0,C 180,E1 18600.738,E2 18600.738} C_VEL
LIN {X 0,Y 389.815,Z 758.637,A -85,B 0,C 180,E1 18598.276,E2 18598.276} C_VEL
LIN {X 0,Y 393.04,Z 741.826,A -85,B 0,C 180,E1 18596.143,E2 18596.143} C_VEL
LIN {X 0,Y 396.356,Z 723.315,A -85,B 0,C 180,E1 18594.179,E2 18594.179} C_VEL
LIN {X 0,Y 399.737,Z 702.918,A -85,B 0,C 180,E1 18592.387,E2 18592.387} C_VEL
LIN {X 0,Y 403.351,Z 679.808,A -85,B 0,C 180,E1 18590.692,E2 18590.692} C_VEL
LIN {X 0,Y 406.75,Z 656.598,A -85,B 0,C 180,E1 18589.305,E2 18589.305} C_VEL
LIN {X 0,Y 409.935,Z 632.544,A -85,B 0,C 180,E1 18588.157,E2 18588.157} C_VEL
LIN {X 0,Y 412.919,Z 607.029,A -85,B 0,C 180,E1 18587.235,E2 18587.235} C_VEL
LIN {X 0,Y 415.18,Z 580.238,A -85,B 0,C 180,E1 18586.509,E2 18586.509} C_VEL
LIN {X 0,Y 416.504,Z 563.71,A -85,B 0,C 180,E1 18586.213,E2 18586.213} C_VEL
LIN {X 0,Y 419.455,Z 541.816,A -85,B 0,C 180,E1 18586.07,E2 18586.07} C_VEL
LIN {X 0,Y 421.286,Z 532.132,A -85,B 0,C 180,E1 18586.036,E2 18586.036} C_VEL
LIN {X 0,Y 430.153,Z 515.586,A -85,B 0,C 180,E1 18585.226,E2 18585.226} C_VEL
LIN {X 0,Y 436.988,Z 504.442,A -85,B 0,C 180,E1 18584.777,E2 18584.777} C_VEL
LIN {X 0,Y 428.558,Z 491.653,A -85,B 0,C 180,E1 18582.699,E2 18582.699} C_VEL
LIN {X 0,Y 421.956,Z 477.021,A -85,B 0,C 180,E1 18580.479,E2 18580.479} C_VEL
LIN {X 0,Y 417.686,Z 461.674,A -85,B 0,C 180,E1 18578.315,E2 18578.315} C_VEL
LIN {X 0,Y 415.381,Z 444.046,A -85,B 0,C 180,E1 18576.022,E2 18576.022} C_VEL
LIN {X 0,Y 415.282,Z 425.307,A -85,B 0,C 180,E1 18573.791,E2 18573.791} C_VEL
LIN {X 0,Y 417.496,Z 404.063,A -85,B 0,C 180,E1 18571.505,E2 18571.505} C_VEL
LIN {X 0,Y 420.235,Z 387.417,A -85,B 0,C 180,E1 18569.819,E2 18569.819} C_VEL
LIN {X 0,Y 409.322,Z 392.341,A -85,B 0,C 180,E1 18568.605,E2 18568.605} C_VEL
LIN {X 0,Y 404.347,Z 394.619,A -85,B 0,C 180,E1 18568.023,E2 18568.023} C_VEL
LIN {X 0,Y 400.124,Z 396.71,A -85,B 0,C 180,E1 18567.535,E2 18567.535} C_VEL
LIN {X 0,Y 398.343,Z 397.472,A -85,B 0,C 180,E1 18567.307,E2 18567.307} C_VEL
LIN {X 0,Y 395.058,Z 399.289,A -85,B 0,C 180,E1 18566.938,E2 18566.938} C_VEL
LIN {X 0,Y 393.166,Z 399.75,A -85,B 0,C 180,E1 18566.588,E2 18566.588} C_VEL
LIN {X 0,Y 391.364,Z 448.508,A -85,B 0,C 180,E1 18562.691,E2 18562.691} C_VEL
LIN {X 0,Y 389.502,Z 496.332,A -85,B 0,C 180,E1 18558.793,E2 18558.793} C_VEL
LIN {X 0,Y 388.696,Z 511.181,A -85,B 0,C 180,E1 18557.592,E2 18557.592} C_VEL
LIN {X 0,Y 386.506,Z 523.718,A -85,B 0,C 180,E1 18556.764,E2 18556.764} C_VEL
LIN {X 0,Y 383.693,Z 618.952,A -85,B 0,C 180,E1 18554.421,E2 18554.421} C_VEL
LIN {X 0,Y 383.771,Z 638.721,A -85,B 0,C 180,E1 18553.858,E2 18553.858} C_VEL
LIN {X 0,Y 383.654,Z 653.12,A -85,B 0,C 180,E1 18553.181,E2 18553.181} C_VEL
LIN {X 0,Y 383.283,Z 666.709,A -85,B 0,C 180,E1 18552.275,E2 18552.275} C_VEL
LIN {X 0,Y 382.723,Z 680.044,A -85,B 0,C 180,E1 18551.07,E2 18551.07} C_VEL
LIN {X 0,Y 382.015,Z 692.084,A -85,B 0,C 180,E1 18549.642,E2 18549.642} C_VEL
LIN {X 0,Y 381.231,Z 702.821,A -85,B 0,C 180,E1 18547.99,E2 18547.99} C_VEL
LIN {X 0,Y 380.456,Z 711.768,A -85,B 0,C 180,E1 18546.185,E2 18546.185} C_VEL
LIN {X 0,Y 379.786,Z 718.549,A -85,B 0,C 180,E1 18544.378,E2 18544.378} C_VEL
LIN {X 0,Y 379.203,Z 723.947,A -85,B 0,C 180,E1 18542.417,E2 18542.417} C_VEL
LIN {X 0,Y 378.725,Z 727.758,A -85,B 0,C 180,E1 18540.302,E2 18540.302} C_VEL
LIN {X 0,Y 378.397,Z 729.676,A -85,B 0,C 180,E1 18538.182,E2 18538.182} C_VEL
LIN {X 0,Y 378.19,Z 729.831,A -85,B 0,C 180,E1 18536.058,E2 18536.058} C_VEL
LIN {X 0,Y 378.112,Z 728.158,A -85,B 0,C 180,E1 18533.871,E2 18533.871} C_VEL
LIN {X 0,Y 378.162,Z 724.494,A -85,B 0,C 180,E1 18531.638,E2 18531.638} C_VEL
LIN {X 0,Y 378.373,Z 718.783,A -85,B 0,C 180,E1 18529.429,E2 18529.429} C_VEL
LIN {X 0,Y 378.73,Z 711.21,A -85,B 0,C 180,E1 18527.342,E2 18527.342} C_VEL
LIN {X 0,Y 379.199,Z 702.359,A -85,B 0,C 180,E1 18525.493,E2 18525.493} C_VEL
LIN {X 0,Y 379.741,Z 691.961,A -85,B 0,C 180,E1 18523.793,E2 18523.793} C_VEL
LIN {X 0,Y 380.309,Z 680.429,A -85,B 0,C 180,E1 18522.307,E2 18522.307} C_VEL
LIN {X 0,Y 380.85,Z 667.484,A -85,B 0,C 180,E1 18521.001,E2 18521.001} C_VEL
LIN {X 0,Y 381.332,Z 653.257,A -85,B 0,C 180,E1 18519.91,E2 18519.91} C_VEL
LIN {X 0,Y 381.648,Z 637.334,A -85,B 0,C 180,E1 18519.039,E2 18519.039} C_VEL
LIN {X 0,Y 381.75,Z 621.063,A -85,B 0,C 180,E1 18518.478,E2 18518.478} C_VEL
LIN {X 0,Y 383.819,Z 509.425,A -85,B 0,C 180,E1 18516.001,E2 18516.001} C_VEL
LIN {X 0,Y 384.697,Z 501.325,A -85,B 0,C 180,E1 18515.344,E2 18515.344} C_VEL
LIN {X 0,Y 386.618,Z 451.59,A -85,B 0,C 180,E1 18511.134,E2 18511.134} C_VEL
LIN {X 0,Y 388.549,Z 404.314,A -85,B 0,C 180,E1 18507.113,E2 18507.113} C_VEL
LIN {X 0,Y 390.469,Z 358.362,A -85,B 0,C 180,E1 18503.187,E2 18503.187} C_VEL
LIN {X 0,Y 390.81,Z 350.93,A -85,B 0,C 180,E1 18502.535,E2 18502.535} C_VEL
LIN {X 0,Y 392.457,Z 350.681,A -85,B 0,C 180,E1 18502.12,E2 18502.12} C_VEL
LIN {X 0,Y 395.177,Z 349.098,A -85,B 0,C 180,E1 18501.691,E2 18501.691} C_VEL
LIN {X 0,Y 396.594,Z 348.219,A -85,B 0,C 180,E1 18501.485,E2 18501.485} C_VEL
LIN {X 0,Y 399.75,Z 346.806,A -85,B 0,C 180,E1 18500.927,E2 18500.927} C_VEL
LIN {X 0,Y 402.509,Z 345.268,A -85,B 0,C 180,E1 18500.511,E2 18500.511} C_VEL
LIN {X 0,Y 415.617,Z 338.983,A -85,B 0,C 180,E1 18498.503,E2 18498.503} C_VEL
LIN {X 0,Y 419.886,Z 349.769,A -85,B 0,C 180,E1 18495.827,E2 18495.827} C_VEL
LIN {X 0,Y 420.872,Z 351.559,A -85,B 0,C 180,E1 18495.641,E2 18495.641} C_VEL
LIN {X 0,Y 417.72,Z 425.006,A -85,B 0,C 180,E1 18494.234,E2 18494.234} C_VEL
LIN {X 0,Y 413.555,Z 491.588,A -85,B 0,C 180,E1 18492.744,E2 18492.744} C_VEL
LIN {X 0,Y 407.822,Z 566.328,A -85,B 0,C 180,E1 18490.802,E2 18490.802} C_VEL
LIN {X 0,Y 405.779,Z 593.893,A -85,B 0,C 180,E1 18489.927,E2 18489.927} C_VEL
LIN {X 0,Y 403.832,Z 614.146,A -85,B 0,C 180,E1 18489.014,E2 18489.014} C_VEL
LIN {X 0,Y 402.285,Z 627.038,A -85,B 0,C 180,E1 18488.286,E2 18488.286} C_VEL
LIN {X 0,Y 400.566,Z 634.229,A -85,B 0,C 180,E1 18487.919,E2 18487.919} C_VEL
LIN {X 0,Y 393.085,Z 652.175,A -85,B 0,C 180,E1 18487.136,E2 18487.136} C_VEL
LIN {X 0,Y 391.169,Z 658.775,A -85,B 0,C 180,E1 18486.659,E2 18486.659} C_VEL
LIN {X 0,Y 388.037,Z 676.011,A -85,B 0,C 180,E1 18484.975,E2 18484.975} C_VEL
LIN {X 0,Y 384.751,Z 692.622,A -85,B 0,C 180,E1 18483.018,E2 18483.018} C_VEL
LIN {X 0,Y 381.523,Z 708.004,A -85,B 0,C 180,E1 18480.849,E2 18480.849} C_VEL
LIN {X 0,Y 378.602,Z 721.65,A -85,B 0,C 180,E1 18478.556,E2 18478.556} C_VEL
LIN {X 0,Y 375.747,Z 735.002,A -85,B 0,C 180,E1 18475.875,E2 18475.875} C_VEL
LIN {X 0,Y 373.453,Z 746.166,A -85,B 0,C 180,E1 18473.177,E2 18473.177} C_VEL
LIN {X 0,Y 371.498,Z 756.453,A -85,B 0,C 180,E1 18470.152,E2 18470.152} C_VEL
LIN {X 0,Y 370.12,Z 764.711,A -85,B 0,C 180,E1 18467.125,E2 18467.125} C_VEL
LIN {X 0,Y 369.178,Z 771.465,A -85,B 0,C 180,E1 18463.948,E2 18463.948} C_VEL
LIN {X 0,Y 368.666,Z 776.39,A -85,B 0,C 180,E1 18460.786,E2 18460.786} C_VEL
LIN {X 0,Y 368.412,Z 779.497,A -85,B 0,C 180,E1 18457.799,E2 18457.799} C_VEL
LIN {X 0,Y 368.314,Z 781.16,A -85,B 0,C 180,E1 18454.671,E2 18454.671} C_VEL
LIN {X 0,Y 368.301,Z 781.164,A -85,B 0,C 180,E1 18451.556,E2 18451.556} C_VEL
LIN {X 0,Y 368.368,Z 779.66,A -85,B 0,C 180,E1 18448.6,E2 18448.6} C_VEL
LIN {X 0,Y 368.584,Z 776.528,A -85,B 0,C 180,E1 18445.488,E2 18445.488} C_VEL
LIN {X 0,Y 369.042,Z 771.732,A -85,B 0,C 180,E1 18442.371,E2 18442.371} C_VEL
LIN {X 0,Y 369.855,Z 765.165,A -85,B 0,C 180,E1 18439.249,E2 18439.249} C_VEL
LIN {X 0,Y 371.09,Z 757.161,A -85,B 0,C 180,E1 18436.284,E2 18436.284} C_VEL
LIN {X 0,Y 372.725,Z 747.821,A -85,B 0,C 180,E1 18433.48,E2 18433.48} C_VEL
LIN {X 0,Y 374.884,Z 736.509,A -85,B 0,C 180,E1 18430.687,E2 18430.687} C_VEL
LIN {X 0,Y 377.442,Z 723.724,A -85,B 0,C 180,E1 18428.067,E2 18428.067} C_VEL
LIN {X 0,Y 380.334,Z 709.426,A -85,B 0,C 180,E1 18425.623,E2 18425.623} C_VEL
LIN {X 0,Y 383.325,Z 694.4,A -85,B 0,C 180,E1 18423.468,E2 18423.468} C_VEL
LIN {X 0,Y 386.437,Z 677.897,A -85,B 0,C 180,E1 18421.489,E2 18421.489} C_VEL
LIN {X 0,Y 389.549,Z 659.974,A -85,B 0,C 180,E1 18419.711,E2 18419.711} C_VEL
LIN {X 0,Y 392.466,Z 640.976,A -85,B 0,C 180,E1 18418.173,E2 18418.173} C_VEL
LIN {X 0,Y 395.042,Z 621.397,A -85,B 0,C 180,E1 18416.906,E2 18416.906} C_VEL
LIN {X 0,Y 397.159,Z 601.286,A -85,B 0,C 180,E1 18415.898,E2 18415.898} C_VEL
LIN {X 0,Y 398.786,Z 580.355,A -85,B 0,C 180,E1 18415.129,E2 18415.129} C_VEL
LIN {X 0,Y 404.319,Z 508.513,A -85,B 0,C 180,E1 18413.163,E2 18413.163} C_VEL
LIN {X 0,Y 408.735,Z 441.679,A -85,B 0,C 180,E1 18411.591,E2 18411.591} C_VEL
LIN {X 0,Y 411.7,Z 380.113,A -85,B 0,C 180,E1 18410.351,E2 18410.351} C_VEL
LIN {X 0,Y 412.726,Z 349.604,A -85,B 0,C 180,E1 18409.767,E2 18409.767} C_VEL
LIN {X 0,Y 412.052,Z 348.527,A -85,B 0,C 180,E1 18409.617,E2 18409.617} C_VEL
LIN {X 0,Y 406.128,Z 334.406,A -85,B 0,C 180,E1 18406.575,E2 18406.575} C_VEL
LIN {X 0,Y 400.007,Z 320.809,A -85,B 0,C 180,E1 18403.228,E2 18403.228} C_VEL
LIN {X 0,Y 393.655,Z 307.941,A -85,B 0,C 180,E1 18399.514,E2 18399.514} C_VEL
LIN {X 0,Y 388.585,Z 298.471,A -85,B 0,C 180,E1 18396.286,E2 18396.286} C_VEL
LIN {X 0,Y 388.28,Z 298.199,A -85,B 0,C 180,E1 18396.136,E2 18396.136} C_VEL
LIN {X 0,Y 383.866,Z 299.539,A -85,B 0,C 180,E1 18394.963,E2 18394.963} C_VEL
LIN {X 0,Y 382.014,Z 300.023,A -85,B 0,C 180,E1 18394.427,E2 18394.427} C_VEL
LIN {X 0,Y 381.738,Z 299.984,A -85,B 0,C 180,E1 18394.296,E2 18394.296} C_VEL
LIN {X 0,Y 385.67,Z 312.707,A -85,B 0,C 180,E1 18392.73,E2 18392.73} C_VEL
LIN {X 0,Y 383.916,Z 354.073,A -85,B 0,C 180,E1 18388.898,E2 18388.898} C_VEL
LIN {X 0,Y 381.932,Z 397.869,A -85,B 0,C 180,E1 18384.868,E2 18384.868} C_VEL
LIN {X 0,Y 379.933,Z 443.198,A -85,B 0,C 180,E1 18380.73,E2 18380.73} C_VEL
LIN {X 0,Y 379.084,Z 460.927,A -85,B 0,C 180,E1 18379.156,E2 18379.156} C_VEL
LIN {X 0,Y 375.655,Z 602.826,A -85,B 0,C 180,E1 18375.852,E2 18375.852} C_VEL
LIN {X 0,Y 375.398,Z 619.97,A -85,B 0,C 180,E1 18375.22,E2 18375.22} C_VEL
LIN {X 0,Y 374.932,Z 635.953,A -85,B 0,C 180,E1 18374.36,E2 18374.36} C_VEL
LIN {X 0,Y 374.275,Z 651.86,A -85,B 0,C 180,E1 18373.204,E2 18373.204} C_VEL
LIN {X 0,Y 373.531,Z 666.555,A -85,B 0,C 180,E1 18371.817,E2 18371.817} C_VEL
LIN {X 0,Y 372.777,Z 679.631,A -85,B 0,C 180,E1 18370.275,E2 18370.275} C_VEL
LIN {X 0,Y 371.962,Z 692.642,A -85,B 0,C 180,E1 18368.347,E2 18368.347} C_VEL
LIN {X 0,Y 371.297,Z 703.365,A -85,B 0,C 180,E1 18366.339,E2 18366.339} C_VEL
LIN {X 0,Y 370.821,Z 711.968,A -85,B 0,C 180,E1 18364.33,E2 18364.33} C_VEL
LIN {X 0,Y 370.461,Z 719.608,A -85,B 0,C 180,E1 18362.011,E2 18362.011} C_VEL
LIN {X 0,Y 370.291,Z 724.933,A -85,B 0,C 180,E1 18359.846,E2 18359.846} C_VEL
LIN {X 0,Y 370.258,Z 729.03,A -85,B 0,C 180,E1 18357.369,E2 18357.369} C_VEL
LIN {X 0,Y 370.381,Z 731.048,A -85,B 0,C 180,E1 18355.045,E2 18355.045} C_VEL
LIN {X 0,Y 370.635,Z 731.364,A -85,B 0,C 180,E1 18352.716,E2 18352.716} C_VEL
LIN {X 0,Y 371.039,Z 729.873,A -85,B 0,C 180,E1 18350.383,E2 18350.383} C_VEL
LIN {X 0,Y 371.617,Z 726.57,A -85,B 0,C 180,E1 18348.044,E2 18348.044} C_VEL
LIN {X 0,Y 372.311,Z 721.477,A -85,B 0,C 180,E1 18345.811,E2 18345.811} C_VEL
LIN {X 0,Y 373.186,Z 714.685,A -85,B 0,C 180,E1 18343.661,E2 18343.661} C_VEL
LIN {X 0,Y 374.158,Z 706.034,A -85,B 0,C 180,E1 18341.62,E2 18341.62} C_VEL
LIN {X 0,Y 375.149,Z 696.21,A -85,B 0,C 180,E1 18339.81,E2 18339.81} C_VEL
LIN {X 0,Y 376.205,Z 684.17,A -85,B 0,C 180,E1 18338.058,E2 18338.058} C_VEL
LIN {X 0,Y 377.129,Z 670.745,A -85,B 0,C 180,E1 18336.54,E2 18336.54} C_VEL
LIN {X 0,Y 377.872,Z 656.654,A -85,B 0,C 180,E1 18335.288,E2 18335.288} C_VEL
LIN {X 0,Y 378.435,Z 641.135,A -85,B 0,C 180,E1 18334.239,E2 18334.239} C_VEL
LIN {X 0,Y 378.736,Z 623.859,A -85,B 0,C 180,E1 18333.408,E2 18333.408} C_VEL
LIN {X 0,Y 378.844,Z 601.042,A -85,B 0,C 180,E1 18332.706,E2 18332.706} C_VEL
LIN {X 0,Y 381.701,Z 532.926,A -85,B 0,C 180,E1 18330.842,E2 18330.842} C_VEL
LIN {X 0,Y 384.672,Z 482.478,A -85,B 0,C 180,E1 18329.373,E2 18329.373} C_VEL
LIN {X 0,Y 387.97,Z 467.508,A -85,B 0,C 180,E1 18328.369,E2 18328.369} C_VEL
LIN {X 0,Y 389.62,Z 440.512,A -85,B 0,C 180,E1 18325.939,E2 18325.939} C_VEL
LIN {X 0,Y 392.478,Z 440.138,A -85,B 0,C 180,E1 18325.56,E2 18325.56} C_VEL
LIN {X 0,Y 396.236,Z 438.122,A -85,B 0,C 180,E1 18325.23,E2 18325.23} C_VEL
LIN {X 0,Y 400.53,Z 436.581,A -85,B 0,C 180,E1 18324.785,E2 18324.785} C_VEL
LIN {X 0,Y 403.252,Z 435.347,A -85,B 0,C 180,E1 18324.536,E2 18324.536} C_VEL
LIN {X 0,Y 417.078,Z 430.042,A -85,B 0,C 180,E1 18323.238,E2 18323.238} C_VEL
LIN {X 0,Y 421.338,Z 446.099,A -85,B 0,C 180,E1 18321.209,E2 18321.209} C_VEL
LIN {X 0,Y 427.735,Z 461.397,A -85,B 0,C 180,E1 18319.117,E2 18319.117} C_VEL
LIN {X 0,Y 435.507,Z 474.547,A -85,B 0,C 180,E1 18317.19,E2 18317.19} C_VEL
LIN {X 0,Y 438.601,Z 479.104,A -85,B 0,C 180,E1 18316.511,E2 18316.511} C_VEL
LIN {X 0,Y 427.271,Z 501.305,A -85,B 0,C 180,E1 18315.732,E2 18315.732} C_VEL
LIN {X 0,Y 418.166,Z 519.423,A -85,B 0,C 180,E1 18315.053,E2 18315.053} C_VEL
LIN {X 0,Y 413.317,Z 531.149,A -85,B 0,C 180,E1 18314.551,E2 18314.551} C_VEL
LIN {X 0,Y 409.953,Z 554.778,A -85,B 0,C 180,E1 18314.414,E2 18314.414} C_VEL
LIN {X 0,Y 408.116,Z 574.924,A -85,B 0,C 180,E1 18314.124,E2 18314.124} C_VEL
LIN {X 0,Y 405.955,Z 602.976,A -85,B 0,C 180,E1 18313.389,E2 18313.389} C_VEL
LIN {X 0,Y 402.837,Z 629.781,A -85,B 0,C 180,E1 18312.441,E2 18312.441} C_VEL
LIN {X 0,Y 399.74,Z 653.69,A -85,B 0,C 180,E1 18311.326,E2 18311.326} C_VEL
LIN {X 0,Y 396.306,Z 677.328,A -85,B 0,C 180,E1 18309.939,E2 18309.939} C_VEL
LIN {X 0,Y 392.629,Z 700.892,A -85,B 0,C 180,E1 18308.23,E2 18308.23} C_VEL
LIN {X 0,Y 389.132,Z 721.785,A -85,B 0,C 180,E1 18306.409,E2 18306.409} C_VEL
LIN {X 0,Y 385.892,Z 739.799,A -85,B 0,C 180,E1 18304.519,E2 18304.519} C_VEL
LIN {X 0,Y 382.623,Z 756.752,A -85,B 0,C 180,E1 18302.392,E2 18302.392} C_VEL
LIN {X 0,Y 379.355,Z 772.84,A -85,B 0,C 180,E1 18299.965,E2 18299.965} C_VEL
LIN {X 0,Y 376.39,Z 787.363,A -85,B 0,C 180,E1 18297.359,E2 18297.359} C_VEL
LIN {X 0,Y 373.626,Z 801.339,A -85,B 0,C 180,E1 18294.338,E2 18294.338} C_VEL
LIN {X 0,Y 371.515,Z 812.921,A -85,B 0,C 180,E1 18291.305,E2 18291.305} C_VEL
LIN {X 0,Y 369.928,Z 822.983,A -85,B 0,C 180,E1 18288.109,E2 18288.109} C_VEL
LIN {X 0,Y 368.871,Z 831.407,A -85,B 0,C 180,E1 18284.762,E2 18284.762} C_VEL
LIN {X 0,Y 368.323,Z 837.838,A -85,B 0,C 180,E1 18281.486,E2 18281.486} C_VEL
LIN {X 0,Y 368.114,Z 842.705,A -85,B 0,C 180,E1 18278.12,E2 18278.12} C_VEL
LIN {X 0,Y 368.091,Z 845.691,A -85,B 0,C 180,E1 18274.987,E2 18274.987} C_VEL
LIN {X 0,Y 368.115,Z 847.267,A -85,B 0,C 180,E1 18271.712,E2 18271.712} C_VEL
LIN {X 0,Y 368.12,Z 847.343,A -85,B 0,C 180,E1 18268.599,E2 18268.599} C_VEL
LIN {X 0,Y 368.097,Z 845.863,A -85,B 0,C 180,E1 18265.326,E2 18265.326} C_VEL
LIN {X 0,Y 368.111,Z 842.845,A -85,B 0,C 180,E1 18262.037,E2 18262.037} C_VEL
LIN {X 0,Y 368.302,Z 838.129,A -85,B 0,C 180,E1 18258.728,E2 18258.728} C_VEL
LIN {X 0,Y 368.833,Z 831.721,A -85,B 0,C 180,E1 18255.397,E2 18255.397} C_VEL
LIN {X 0,Y 369.925,Z 822.965,A -85,B 0,C 180,E1 18251.891,E2 18251.891} C_VEL
LIN {X 0,Y 371.52,Z 812.99,A -85,B 0,C 180,E1 18248.695,E2 18248.695} C_VEL
LIN {X 0,Y 373.635,Z 801.54,A -85,B 0,C 180,E1 18245.662,E2 18245.662} C_VEL
LIN {X 0,Y 376.418,Z 787.723,A -85,B 0,C 180,E1 18242.643,E2 18242.643} C_VEL
LIN {X 0,Y 379.415,Z 773.477,A -85,B 0,C 180,E1 18240.04,E2 18240.04} C_VEL
LIN {X 0,Y 382.881,Z 756.916,A -85,B 0,C 180,E1 18237.509,E2 18237.509} C_VEL
LIN {X 0,Y 386.157,Z 740.569,A -85,B 0,C 180,E1 18235.424,E2 18235.424} C_VEL
LIN {X 0,Y 389.664,Z 721.849,A -85,B 0,C 180,E1 18233.431,E2 18233.431} C_VEL
LIN {X 0,Y 393.171,Z 701.55,A -85,B 0,C 180,E1 18231.646,E2 18231.646} C_VEL
LIN {X 0,Y 396.928,Z 678.505,A -85,B 0,C 180,E1 18229.948,E2 18229.948} C_VEL
LIN {X 0,Y 400.433,Z 655.558,A -85,B 0,C 180,E1 18228.571,E2 18228.571} C_VEL
LIN {X 0,Y 403.853,Z 630.679,A -85,B 0,C 180,E1 18227.38,E2 18227.38} C_VEL
LIN {X 0,Y 407,Z 604.86,A -85,B 0,C 180,E1 18226.45,E2 18226.45} C_VEL
LIN {X 0,Y 409.342,Z 577.69,A -85,B 0,C 180,E1 18225.71,E2 18225.71} C_VEL
LIN {X 0,Y 410.873,Z 561.251,A -85,B 0,C 180,E1 18225.441,E2 18225.441} C_VEL
LIN {X 0,Y 413.848,Z 539.967,A -85,B 0,C 180,E1 18225.317,E2 18225.317} C_VEL
LIN {X 0,Y 415.707,Z 529.841,A -85,B 0,C 180,E1 18225.289,E2 18225.289} C_VEL
LIN {X 0,Y 424.72,Z 513.334,A -85,B 0,C 180,E1 18224.495,E2 18224.495} C_VEL
LIN {X 0,Y 428.707,Z 506.657,A -85,B 0,C 180,E1 18224.214,E2 18224.214} C_VEL
LIN {X 0,Y 421.148,Z 494.334,A -85,B 0,C 180,E1 18222.206,E2 18222.206} C_VEL
LIN {X 0,Y 414.76,Z 479.137,A -85,B 0,C 180,E1 18219.884,E2 18219.884} C_VEL
LIN {X 0,Y 410.824,Z 463.411,A -85,B 0,C 180,E1 18217.653,E2 18217.653} C_VEL
LIN {X 0,Y 408.893,Z 445.702,A -85,B 0,C 180,E1 18215.331,E2 18215.331} C_VEL
LIN {X 0,Y 409.15,Z 426.427,A -85,B 0,C 180,E1 18213.021,E2 18213.021} C_VEL
LIN {X 0,Y 411.804,Z 404.553,A -85,B 0,C 180,E1 18210.655,E2 18210.655} C_VEL
LIN {X 0,Y 413.158,Z 396.468,A -85,B 0,C 180,E1 18209.822,E2 18209.822} C_VEL
LIN {X 0,Y 402.569,Z 401.367,A -85,B 0,C 180,E1 18208.643,E2 18208.643} C_VEL
LIN {X 0,Y 396.655,Z 404.222,A -85,B 0,C 180,E1 18207.96,E2 18207.96} C_VEL
LIN {X 0,Y 391.663,Z 406.601,A -85,B 0,C 180,E1 18207.355,E2 18207.355} C_VEL
LIN {X 0,Y 388.16,Z 408.546,A -85,B 0,C 180,E1 18206.959,E2 18206.959} C_VEL
LIN {X 0,Y 386.345,Z 408.972,A -85,B 0,C 180,E1 18206.618,E2 18206.618} C_VEL
LIN {X 0,Y 384.354,Z 455.959,A -85,B 0,C 180,E1 18202.805,E2 18202.805} C_VEL
LIN {X 0,Y 382.309,Z 503.977,A -85,B 0,C 180,E1 18198.836,E2 18198.836} C_VEL
LIN {X 0,Y 381.745,Z 512.366,A -85,B 0,C 180,E1 18198.16,E2 18198.16} C_VEL
LIN {X 0,Y 379.393,Z 525.388,A -85,B 0,C 180,E1 18197.291,E2 18197.291} C_VEL
LIN {X 0,Y 376.363,Z 616.77,A -85,B 0,C 180,E1 18194.957,E2 18194.957} C_VEL
LIN {X 0,Y 376.385,Z 639.745,A -85,B 0,C 180,E1 18194.297,E2 18194.297} C_VEL
LIN {X 0,Y 376.24,Z 654.578,A -85,B 0,C 180,E1 18193.586,E2 18193.586} C_VEL
LIN {X 0,Y 375.842,Z 667.935,A -85,B 0,C 180,E1 18192.678,E2 18192.678} C_VEL
LIN {X 0,Y 375.245,Z 681.378,A -85,B 0,C 180,E1 18191.449,E2 18191.449} C_VEL
LIN {X 0,Y 374.484,Z 693.471,A -85,B 0,C 180,E1 18189.994,E2 18189.994} C_VEL
LIN {X 0,Y 373.631,Z 704.208,A -85,B 0,C 180,E1 18188.308,E2 18188.308} C_VEL
LIN {X 0,Y 372.793,Z 713.175,A -85,B 0,C 180,E1 18186.467,E2 18186.467} C_VEL
LIN {X 0,Y 372.069,Z 719.987,A -85,B 0,C 180,E1 18184.624,E2 18184.624} C_VEL
LIN {X 0,Y 371.435,Z 725.392,A -85,B 0,C 180,E1 18182.622,E2 18182.622} C_VEL
LIN {X 0,Y 370.907,Z 729.181,A -85,B 0,C 180,E1 18180.463,E2 18180.463} C_VEL
LIN {X 0,Y 370.541,Z 731.074,A -85,B 0,C 180,E1 18178.299,E2 18178.299} C_VEL
LIN {X 0,Y 370.31,Z 731.209,A -85,B 0,C 180,E1 18176.129,E2 18176.129} C_VEL
LIN {X 0,Y 370.217,Z 729.561,A -85,B 0,C 180,E1 18173.953,E2 18173.953} C_VEL
LIN {X 0,Y 370.26,Z 725.77,A -85,B 0,C 180,E1 18171.614,E2 18171.614} C_VEL
LIN {X 0,Y 370.466,Z 720.186,A -85,B 0,C 180,E1 18169.424,E2 18169.424} C_VEL
LIN {X 0,Y 370.808,Z 712.976,A -85,B 0,C 180,E1 18167.384,E2 18167.384} C_VEL
LIN {X 0,Y 371.285,Z 704.232,A -85,B 0,C 180,E1 18165.495,E2 18165.495} C_VEL
LIN {X 0,Y 371.84,Z 693.971,A -85,B 0,C 180,E1 18163.76,E2 18163.76} C_VEL
LIN {X 0,Y 372.447,Z 682.07,A -85,B 0,C 180,E1 18162.179,E2 18162.179} C_VEL
LIN {X 0,Y 373.018,Z 669.032,A -85,B 0,C 180,E1 18160.828,E2 18160.828} C_VEL
LIN {X 0,Y 373.518,Z 654.838,A -85,B 0,C 180,E1 18159.711,E2 18159.711} C_VEL
LIN {X 0,Y 373.858,Z 638.933,A -85,B 0,C 180,E1 18158.813,E2 18158.813} C_VEL
LIN {X 0,Y 373.975,Z 622.491,A -85,B 0,C 180,E1 18158.227,E2 18158.227} C_VEL
LIN {X 0,Y 376.113,Z 510.736,A -85,B 0,C 180,E1 18155.689,E2 18155.689} C_VEL
LIN {X 0,Y 377.1,Z 502.068,A -85,B 0,C 180,E1 18154.981,E2 18154.981} C_VEL
LIN {X 0,Y 379.132,Z 451.794,A -85,B 0,C 180,E1 18150.686,E2 18150.686} C_VEL
LIN {X 0,Y 381.133,Z 404.859,A -85,B 0,C 180,E1 18146.66,E2 18146.66} C_VEL
LIN {X 0,Y 383.152,Z 360.225,A -85,B 0,C 180,E1 18142.787,E2 18142.787} C_VEL
LIN {X 0,Y 384.805,Z 359.939,A -85,B 0,C 180,E1 18142.365,E2 18142.365} C_VEL
LIN {X 0,Y 387.519,Z 358.331,A -85,B 0,C 180,E1 18141.927,E2 18141.927} C_VEL
LIN {X 0,Y 388.949,Z 357.401,A -85,B 0,C 180,E1 18141.717,E2 18141.717} C_VEL
LIN {X 0,Y 392.099,Z 355.961,A -85,B 0,C 180,E1 18141.148,E2 18141.148} C_VEL
LIN {X 0,Y 394.892,Z 354.33,A -85,B 0,C 180,E1 18140.728,E2 18140.728} C_VEL
LIN {X 0,Y 410.873,Z 346.438,A -85,B 0,C 180,E1 18138.274,E2 18138.274} C_VEL
LIN {X 0,Y 413.369,Z 352.585,A -85,B 0,C 180,E1 18136.728,E2 18136.728} C_VEL
LIN {X 0,Y 415.251,Z 355.353,A -85,B 0,C 180,E1 18136.375,E2 18136.375} C_VEL
LIN {X 0,Y 412.027,Z 426.942,A -85,B 0,C 180,E1 18134.989,E2 18134.989} C_VEL
LIN {X 0,Y 407.814,Z 491.396,A -85,B 0,C 180,E1 18133.528,E2 18133.528} C_VEL
LIN {X 0,Y 401.996,Z 563.616,A -85,B 0,C 180,E1 18131.625,E2 18131.625} C_VEL
LIN {X 0,Y 399.584,Z 594.419,A -85,B 0,C 180,E1 18130.645,E2 18130.645} C_VEL
LIN {X 0,Y 397.603,Z 614.288,A -85,B 0,C 180,E1 18129.745,E2 18129.745} C_VEL
LIN {X 0,Y 395.138,Z 633.606,A -85,B 0,C 180,E1 18128.605,E2 18128.605} C_VEL
LIN {X 0,Y 392.185,Z 652.818,A -85,B 0,C 180,E1 18127.173,E2 18127.173} C_VEL
LIN {X 0,Y 391.169,Z 658.775,A -85,B 0,C 180,E1 18126.659,E2 18126.659} C_VEL
LIN {X 0,Y 389.218,Z 665.43,A -85,B 0,C 180,E1 18126.144,E2 18126.144} C_VEL
LIN {X 0,Y 381.131,Z 682.018,A -85,B 0,C 180,E1 18124.955,E2 18124.955} C_VEL
LIN {X 0,Y 379.031,Z 688.166,A -85,B 0,C 180,E1 18124.319,E2 18124.319} C_VEL
LIN {X 0,Y 375.556,Z 704.174,A -85,B 0,C 180,E1 18122.152,E2 18122.152} C_VEL
LIN {X 0,Y 372.264,Z 718.713,A -85,B 0,C 180,E1 18119.795,E2 18119.795} C_VEL
LIN {X 0,Y 369.086,Z 732.663,A -85,B 0,C 180,E1 18117.073,E2 18117.073} C_VEL
LIN {X 0,Y 366.356,Z 744.943,A -85,B 0,C 180,E1 18114.166,E2 18114.166} C_VEL
LIN {X 0,Y 364.25,Z 755.101,A -85,B 0,C 180,E1 18111.244,E2 18111.244} C_VEL
LIN {X 0,Y 362.629,Z 763.797,A -85,B 0,C 180,E1 18108.154,E2 18108.154} C_VEL
LIN {X 0,Y 361.495,Z 770.956,A -85,B 0,C 180,E1 18104.906,E2 18104.906} C_VEL
LIN {X 0,Y 360.837,Z 776.254,A -85,B 0,C 180,E1 18101.67,E2 18101.67} C_VEL
LIN {X 0,Y 360.501,Z 779.794,A -85,B 0,C 180,E1 18098.453,E2 18098.453} C_VEL
LIN {X 0,Y 360.359,Z 781.615,A -85,B 0,C 180,E1 18095.413,E2 18095.413} C_VEL
LIN {X 0,Y 360.324,Z 781.975,A -85,B 0,C 180,E1 18092.226,E2 18092.226} C_VEL
LIN {X 0,Y 360.39,Z 780.732,A -85,B 0,C 180,E1 18089.046,E2 18089.046} C_VEL
LIN {X 0,Y 360.577,Z 778.084,A -85,B 0,C 180,E1 18086.025,E2 18086.025} C_VEL
LIN {X 0,Y 361.016,Z 773.67,A -85,B 0,C 180,E1 18082.841,E2 18082.841} C_VEL
LIN {X 0,Y 361.802,Z 767.487,A -85,B 0,C 180,E1 18079.652,E2 18079.652} C_VEL
LIN {X 0,Y 363.118,Z 759.287,A -85,B 0,C 180,E1 18076.412,E2 18076.412} C_VEL
LIN {X 0,Y 364.957,Z 749.285,A -85,B 0,C 180,E1 18073.282,E2 18073.282} C_VEL
LIN {X 0,Y 367.249,Z 737.949,A -85,B 0,C 180,E1 18070.394,E2 18070.394} C_VEL
LIN {X 0,Y 370.051,Z 724.669,A -85,B 0,C 180,E1 18067.606,E2 18067.606} C_VEL
LIN {X 0,Y 373.091,Z 710.415,A -85,B 0,C 180,E1 18065.118,E2 18065.118} C_VEL
LIN {X 0,Y 376.279,Z 695.199,A -85,B 0,C 180,E1 18062.896,E2 18062.896} C_VEL
LIN {X 0,Y 379.618,Z 678.27,A -85,B 0,C 180,E1 18060.839,E2 18060.839} C_VEL
LIN {X 0,Y 382.737,Z 661.161,A -85,B 0,C 180,E1 18059.114,E2 18059.114} C_VEL
LIN {X 0,Y 385.78,Z 642.271,A -85,B 0,C 180,E1 18057.554,E2 18057.554} C_VEL
LIN {X 0,Y 388.468,Z 622.778,A -85,B 0,C 180,E1 18056.268,E2 18056.268} C_VEL
LIN {X 0,Y 390.692,Z 602.647,A -85,B 0,C 180,E1 18055.237,E2 18055.237} C_VEL
LIN {X 0,Y 392.398,Z 581.844,A -85,B 0,C 180,E1 18054.454,E2 18054.454} C_VEL
LIN {X 0,Y 397.941,Z 513.592,A -85,B 0,C 180,E1 18052.534,E2 18052.534} C_VEL
LIN {X 0,Y 402.604,Z 447.168,A -85,B 0,C 180,E1 18050.93,E2 18050.93} C_VEL
LIN {X 0,Y 405.763,Z 385.849,A -85,B 0,C 180,E1 18049.67,E2 18049.67} C_VEL
LIN {X 0,Y 406.939,Z 353.455,A -85,B 0,C 180,E1 18049.046,E2 18049.046} C_VEL
LIN {X 0,Y 405.521,Z 351.273,A -85,B 0,C 180,E1 18048.766,E2 18048.766} C_VEL
LIN {X 0,Y 399.731,Z 337.462,A -85,B 0,C 180,E1 18045.675,E2 18045.675} C_VEL
LIN {X 0,Y 394.407,Z 325.743,A -85,B 0,C 180,E1 18042.677,E2 18042.677} C_VEL
LIN {X 0,Y 388.779,Z 314.055,A -85,B 0,C 180,E1 18039.248,E2 18039.248} C_VEL
LIN {X 0,Y 384.317,Z 305.372,A -85,B 0,C 180,E1 18036.291,E2 18036.291} C_VEL
LIN {X 0,Y 378.113,Z 307.462,A -85,B 0,C 180,E1 18034.649,E2 18034.649} C_VEL
LIN {X 0,Y 376.193,Z 307.827,A -85,B 0,C 180,E1 18034.043,E2 18034.043} C_VEL
LIN {X 0,Y 378.388,Z 315.52,A -85,B 0,C 180,E1 18033.071,E2 18033.071} C_VEL
LIN {X 0,Y 376.473,Z 358.258,A -85,B 0,C 180,E1 18029.08,E2 18029.08} C_VEL
LIN {X 0,Y 374.417,Z 401.802,A -85,B 0,C 180,E1 18025.042,E2 18025.042} C_VEL
LIN {X 0,Y 372.292,Z 447.445,A -85,B 0,C 180,E1 18020.832,E2 18020.832} C_VEL
LIN {X 0,Y 371.52,Z 461.754,A -85,B 0,C 180,E1 18019.546,E2 18019.546} C_VEL
LIN {X 0,Y 367.916,Z 602.971,A -85,B 0,C 180,E1 18016.165,E2 18016.165} C_VEL
LIN {X 0,Y 367.668,Z 619.832,A -85,B 0,C 180,E1 18015.548,E2 18015.548} C_VEL
LIN {X 0,Y 367.158,Z 636.916,A -85,B 0,C 180,E1 18014.623,E2 18014.623} C_VEL
LIN {X 0,Y 366.456,Z 653.254,A -85,B 0,C 180,E1 18013.411,E2 18013.411} C_VEL
LIN {X 0,Y 365.688,Z 667.924,A -85,B 0,C 180,E1 18011.994,E2 18011.994} C_VEL
LIN {X 0,Y 364.911,Z 681.008,A -85,B 0,C 180,E1 18010.419,E2 18010.419} C_VEL
LIN {X 0,Y 364.102,Z 693.574,A -85,B 0,C 180,E1 18008.528,E2 18008.528} C_VEL
LIN {X 0,Y 363.461,Z 703.685,A -85,B 0,C 180,E1 18006.635,E2 18006.635} C_VEL
LIN {X 0,Y 362.926,Z 713.144,A -85,B 0,C 180,E1 18004.425,E2 18004.425} C_VEL
LIN {X 0,Y 362.559,Z 720.882,A -85,B 0,C 180,E1 18002.055,E2 18002.055} C_VEL
LIN {X 0,Y 362.389,Z 726.277,A -85,B 0,C 180,E1 17999.842,E2 17999.842} C_VEL
LIN {X 0,Y 362.369,Z 730.435,A -85,B 0,C 180,E1 17997.312,E2 17997.312} C_VEL
LIN {X 0,Y 362.514,Z 732.502,A -85,B 0,C 180,E1 17994.937,E2 17994.937} C_VEL
LIN {X 0,Y 362.804,Z 732.859,A -85,B 0,C 180,E1 17992.558,E2 17992.558} C_VEL
LIN {X 0,Y 363.254,Z 731.381,A -85,B 0,C 180,E1 17990.175,E2 17990.175} C_VEL
LIN {X 0,Y 363.893,Z 728.093,A -85,B 0,C 180,E1 17987.786,E2 17987.786} C_VEL
LIN {X 0,Y 364.649,Z 723.137,A -85,B 0,C 180,E1 17985.551,E2 17985.551} C_VEL
LIN {X 0,Y 365.54,Z 716.747,A -85,B 0,C 180,E1 17983.473,E2 17983.473} C_VEL
LIN {X 0,Y 366.594,Z 708.267,A -85,B 0,C 180,E1 17981.392,E2 17981.392} C_VEL
LIN {X 0,Y 367.621,Z 699.112,A -85,B 0,C 180,E1 17979.627,E2 17979.627} C_VEL
LIN {X 0,Y 368.721,Z 687.451,A -85,B 0,C 180,E1 17977.857,E2 17977.857} C_VEL
LIN {X 0,Y 369.682,Z 675.482,A -85,B 0,C 180,E1 17976.404,E2 17976.404} C_VEL
LIN {X 0,Y 370.538,Z 661.255,A -85,B 0,C 180,E1 17975.049,E2 17975.049} C_VEL
LIN {X 0,Y 371.197,Z 646.351,A -85,B 0,C 180,E1 17973.957,E2 17973.957} C_VEL
LIN {X 0,Y 371.595,Z 630.335,A -85,B 0,C 180,E1 17973.088,E2 17973.088} C_VEL
LIN {X 0,Y 371.723,Z 612.515,A -85,B 0,C 180,E1 17972.437,E2 17972.437} C_VEL
LIN {X 0,Y 373.082,Z 570.27,A -85,B 0,C 180,E1 17971.23,E2 17971.23} C_VEL
LIN {X 0,Y 378.213,Z 485.126,A -85,B 0,C 180,E1 17968.704,E2 17968.704} C_VEL
LIN {X 0,Y 381.843,Z 469.03,A -85,B 0,C 180,E1 17967.624,E2 17967.624} C_VEL
LIN {X 0,Y 383.179,Z 449.973,A -85,B 0,C 180,E1 17965.875,E2 17965.875} C_VEL
LIN {X 0,Y 385.628,Z 449.692,A -85,B 0,C 180,E1 17965.54,E2 17965.54} C_VEL
LIN {X 0,Y 390.061,Z 447.412,A -85,B 0,C 180,E1 17965.137,E2 17965.137} C_VEL
LIN {X 0,Y 394.556,Z 445.615,A -85,B 0,C 180,E1 17964.686,E2 17964.686} C_VEL
LIN {X 0,Y 397.153,Z 444.485,A -85,B 0,C 180,E1 17964.44,E2 17964.44} C_VEL
LIN {X 0,Y 409.663,Z 439.43,A -85,B 0,C 180,E1 17963.276,E2 17963.276} C_VEL
LIN {X 0,Y 411.821,Z 438.746,A -85,B 0,C 180,E1 17963.066,E2 17963.066} C_VEL
LIN {X 0,Y 416.813,Z 455.331,A -85,B 0,C 180,E1 17960.885,E2 17960.885} C_VEL
LIN {X 0,Y 424.019,Z 470.847,A -85,B 0,C 180,E1 17958.681,E2 17958.681} C_VEL
LIN {X 0,Y 430.635,Z 481.562,A -85,B 0,C 180,E1 17957.077,E2 17957.077} C_VEL
LIN {X 0,Y 421.03,Z 500.378,A -85,B 0,C 180,E1 17956.412,E2 17956.412} C_VEL
LIN {X 0,Y 411.489,Z 519.424,A -85,B 0,C 180,E1 17955.692,E2 17955.692} C_VEL
LIN {X 0,Y 407.602,Z 528.799,A -85,B 0,C 180,E1 17955.298,E2 17955.298} C_VEL
LIN {X 0,Y 403.966,Z 554.121,A -85,B 0,C 180,E1 17955.157,E2 17955.157} C_VEL
LIN {X 0,Y 402.007,Z 574.464,A -85,B 0,C 180,E1 17954.862,E2 17954.862} C_VEL
LIN {X 0,Y 399.774,Z 601.872,A -85,B 0,C 180,E1 17954.127,E2 17954.127} C_VEL
LIN {X 0,Y 396.459,Z 629.342,A -85,B 0,C 180,E1 17953.145,E2 17953.145} C_VEL
LIN {X 0,Y 393.133,Z 653.866,A -85,B 0,C 180,E1 17951.982,E2 17951.982} C_VEL
LIN {X 0,Y 389.408,Z 678.332,A -85,B 0,C 180,E1 17950.513,E2 17950.513} C_VEL
LIN {X 0,Y 385.748,Z 700.893,A -85,B 0,C 180,E1 17948.849,E2 17948.849} C_VEL
LIN {X 0,Y 382.104,Z 721.747,A -85,B 0,C 180,E1 17947.002,E2 17947.002} C_VEL
LIN {X 0,Y 378.538,Z 740.672,A -85,B 0,C 180,E1 17944.972,E2 17944.972} C_VEL
LIN {X 0,Y 375.186,Z 757.146,A -85,B 0,C 180,E1 17942.842,E2 17942.842} C_VEL
LIN {X 0,Y 371.683,Z 773.658,A -85,B 0,C 180,E1 17940.287,E2 17940.287} C_VEL
LIN {X 0,Y 368.612,Z 787.907,A -85,B 0,C 180,E1 17937.635,E2 17937.635} C_VEL
LIN {X 0,Y 365.89,Z 801.082,A -85,B 0,C 180,E1 17934.715,E2 17934.715} C_VEL
LIN {X 0,Y 363.577,Z 813.166,A -85,B 0,C 180,E1 17931.454,E2 17931.454} C_VEL
LIN {X 0,Y 362.011,Z 822.605,A -85,B 0,C 180,E1 17928.353,E2 17928.353} C_VEL
LIN {X 0,Y 360.905,Z 831.005,A -85,B 0,C 180,E1 17924.931,E2 17924.931} C_VEL
LIN {X 0,Y 360.334,Z 837.451,A -85,B 0,C 180,E1 17921.525,E2 17921.525} C_VEL
LIN {X 0,Y 360.13,Z 842.177,A -85,B 0,C 180,E1 17918.14,E2 17918.14} C_VEL
LIN {X 0,Y 360.119,Z 845.181,A -85,B 0,C 180,E1 17914.778,E2 17914.778} C_VEL
LIN {X 0,Y 360.15,Z 846.637,A -85,B 0,C 180,E1 17911.432,E2 17911.432} C_VEL
LIN {X 0,Y 360.148,Z 846.54,A -85,B 0,C 180,E1 17908.25,E2 17908.25} C_VEL
LIN {X 0,Y 360.119,Z 844.94,A -85,B 0,C 180,E1 17904.903,E2 17904.903} C_VEL
LIN {X 0,Y 360.136,Z 841.947,A -85,B 0,C 180,E1 17901.699,E2 17901.699} C_VEL
LIN {X 0,Y 360.372,Z 836.895,A -85,B 0,C 180,E1 17898.152,E2 17898.152} C_VEL
LIN {X 0,Y 360.984,Z 830.289,A -85,B 0,C 180,E1 17894.744,E2 17894.744} C_VEL
LIN {X 0,Y 362.185,Z 821.581,A -85,B 0,C 180,E1 17891.242,E2 17891.242} C_VEL
LIN {X 0,Y 363.991,Z 811.129,A -85,B 0,C 180,E1 17887.893,E2 17887.893} C_VEL
LIN {X 0,Y 366.329,Z 799.4,A -85,B 0,C 180,E1 17884.799,E2 17884.799} C_VEL
LIN {X 0,Y 369.365,Z 785.304,A -85,B 0,C 180,E1 17881.724,E2 17881.724} C_VEL
LIN {X 0,Y 372.694,Z 770.195,A -85,B 0,C 180,E1 17878.996,E2 17878.996} C_VEL
LIN {X 0,Y 376.263,Z 754.018,A -85,B 0,C 180,E1 17876.553,E2 17876.553} C_VEL
LIN {X 0,Y 379.928,Z 736.392,A -85,B 0,C 180,E1 17874.343,E2 17874.343} C_VEL
LIN {X 0,Y 383.379,Z 718.542,A -85,B 0,C 180,E1 17872.484,E2 17872.484} C_VEL
LIN {X 0,Y 387.202,Z 697.197,A -85,B 0,C 180,E1 17870.634,E2 17870.634} C_VEL
LIN {X 0,Y 391.01,Z 674.599,A -85,B 0,C 180,E1 17869.011,E2 17869.011} C_VEL
LIN {X 0,Y 394.786,Z 650.468,A -85,B 0,C 180,E1 17867.594,E2 17867.594} C_VEL
LIN {X 0,Y 398.356,Z 625.294,A -85,B 0,C 180,E1 17866.437,E2 17866.437} C_VEL
LIN {X 0,Y 401.768,Z 597.045,A -85,B 0,C 180,E1 17865.468,E2 17865.468} C_VEL
LIN {X 0,Y 404.095,Z 570.016,A -85,B 0,C 180,E1 17864.785,E2 17864.785} C_VEL
LIN {X 0,Y 406.945,Z 546.513,A -85,B 0,C 180,E1 17864.562,E2 17864.562} C_VEL
LIN {X 0,Y 410.207,Z 527.56,A -85,B 0,C 180,E1 17864.524,E2 17864.524} C_VEL
LIN {X 0,Y 419.826,Z 510.315,A -85,B 0,C 180,E1 17863.712,E2 17863.712} C_VEL
LIN {X 0,Y 420.555,Z 508.839,A -85,B 0,C 180,E1 17863.634,E2 17863.634} C_VEL
LIN {X 0,Y 413.275,Z 495.885,A -85,B 0,C 180,E1 17861.521,E2 17861.521} C_VEL
LIN {X 0,Y 407.622,Z 481.164,A -85,B 0,C 180,E1 17859.26,E2 17859.26} C_VEL
LIN {X 0,Y 404.039,Z 465.108,A -85,B 0,C 180,E1 17856.966,E2 17856.966} C_VEL
LIN {X 0,Y 402.47,Z 447.102,A -85,B 0,C 180,E1 17854.587,E2 17854.587} C_VEL
LIN {X 0,Y 403.109,Z 427.527,A -85,B 0,C 180,E1 17852.227,E2 17852.227} C_VEL
LIN {X 0,Y 406.043,Z 405.591,A -85,B 0,C 180,E1 17849.829,E2 17849.829} C_VEL
LIN {X 0,Y 395.787,Z 410.433,A -85,B 0,C 180,E1 17848.684,E2 17848.684} C_VEL
LIN {X 0,Y 390.669,Z 412.942,A -85,B 0,C 180,E1 17848.093,E2 17848.093} C_VEL
LIN {X 0,Y 386.413,Z 415.078,A -85,B 0,C 180,E1 17847.591,E2 17847.591} C_VEL
LIN {X 0,Y 384.752,Z 415.871,A -85,B 0,C 180,E1 17847.385,E2 17847.385} C_VEL
LIN {X 0,Y 381.266,Z 417.784,A -85,B 0,C 180,E1 17846.98,E2 17846.98} C_VEL
LIN {X 0,Y 379.628,Z 418.125,A -85,B 0,C 180,E1 17846.683,E2 17846.683} C_VEL
LIN {X 0,Y 377.246,Z 467.497,A -85,B 0,C 180,E1 17842.6,E2 17842.6} C_VEL
LIN {X 0,Y 375.172,Z 511.675,A -85,B 0,C 180,E1 17838.896,E2 17838.896} C_VEL
LIN {X 0,Y 372.346,Z 527.431,A -85,B 0,C 180,E1 17837.84,E2 17837.84} C_VEL
LIN {X 0,Y 369.056,Z 618.867,A -85,B 0,C 180,E1 17835.417,E2 17835.417} C_VEL
LIN {X 0,Y 369.035,Z 641.704,A -85,B 0,C 180,E1 17834.723,E2 17834.723} C_VEL
LIN {X 0,Y 368.888,Z 655.712,A -85,B 0,C 180,E1 17834.039,E2 17834.039} C_VEL
LIN {X 0,Y 368.455,Z 669.396,A -85,B 0,C 180,E1 17833.096,E2 17833.096} C_VEL
LIN {X 0,Y 367.811,Z 682.601,A -85,B 0,C 180,E1 17831.865,E2 17831.865} C_VEL
LIN {X 0,Y 366.972,Z 694.881,A -85,B 0,C 180,E1 17830.359,E2 17830.359} C_VEL
LIN {X 0,Y 366.06,Z 705.673,A -85,B 0,C 180,E1 17828.64,E2 17828.64} C_VEL
LIN {X 0,Y 365.225,Z 713.988,A -85,B 0,C 180,E1 17826.918,E2 17826.918} C_VEL
LIN {X 0,Y 364.428,Z 720.973,A -85,B 0,C 180,E1 17825.036,E2 17825.036} C_VEL
LIN {X 0,Y 363.672,Z 726.844,A -85,B 0,C 180,E1 17822.836,E2 17822.836} C_VEL
LIN {X 0,Y 363.096,Z 730.626,A -85,B 0,C 180,E1 17820.631,E2 17820.631} C_VEL
LIN {X 0,Y 362.691,Z 732.499,A -85,B 0,C 180,E1 17818.42,E2 17818.42} C_VEL
LIN {X 0,Y 362.431,Z 732.586,A -85,B 0,C 180,E1 17816.203,E2 17816.203} C_VEL
LIN {X 0,Y 362.32,Z 730.894,A -85,B 0,C 180,E1 17813.98,E2 17813.98} C_VEL
LIN {X 0,Y 362.357,Z 727.044,A -85,B 0,C 180,E1 17811.59,E2 17811.59} C_VEL
LIN {X 0,Y 362.566,Z 721.386,A -85,B 0,C 180,E1 17809.352,E2 17809.352} C_VEL
LIN {X 0,Y 362.927,Z 713.948,A -85,B 0,C 180,E1 17807.232,E2 17807.232} C_VEL
LIN {X 0,Y 363.413,Z 705.241,A -85,B 0,C 180,E1 17805.337,E2 17805.337} C_VEL
LIN {X 0,Y 363.989,Z 694.852,A -85,B 0,C 180,E1 17803.564,E2 17803.564} C_VEL
LIN {X 0,Y 364.586,Z 683.481,A -85,B 0,C 180,E1 17802.029,E2 17802.029} C_VEL
LIN {X 0,Y 365.176,Z 670.463,A -85,B 0,C 180,E1 17800.652,E2 17800.652} C_VEL
LIN {X 0,Y 365.689,Z 656.345,A -85,B 0,C 180,E1 17799.514,E2 17799.514} C_VEL
LIN {X 0,Y 366.045,Z 640.914,A -85,B 0,C 180,E1 17798.613,E2 17798.613} C_VEL
LIN {X 0,Y 366.184,Z 624.702,A -85,B 0,C 180,E1 17798,E2 17798} C_VEL
LIN {X 0,Y 367.789,Z 537.084,A -85,B 0,C 180,E1 17795.942,E2 17795.942} C_VEL
LIN {X 0,Y 368.529,Z 511.313,A -85,B 0,C 180,E1 17795.302,E2 17795.302} C_VEL
LIN {X 0,Y 369.508,Z 502.837,A -85,B 0,C 180,E1 17794.611,E2 17794.611} C_VEL
LIN {X 0,Y 371.601,Z 453.109,A -85,B 0,C 180,E1 17790.324,E2 17790.324} C_VEL
LIN {X 0,Y 373.737,Z 405.375,A -85,B 0,C 180,E1 17786.188,E2 17786.188} C_VEL
LIN {X 0,Y 375.476,Z 369.614,A -85,B 0,C 180,E1 17783.047,E2 17783.047} C_VEL
LIN {X 0,Y 377.289,Z 369.851,A -85,B 0,C 180,E1 17782.635,E2 17782.635} C_VEL
LIN {X 0,Y 379.876,Z 367.712,A -85,B 0,C 180,E1 17782.173,E2 17782.173} C_VEL
LIN {X 0,Y 381.292,Z 366.681,A -85,B 0,C 180,E1 17781.957,E2 17781.957} C_VEL
LIN {X 0,Y 384.431,Z 365.211,A -85,B 0,C 180,E1 17781.375,E2 17781.375} C_VEL
LIN {X 0,Y 387.241,Z 363.515,A -85,B 0,C 180,E1 17780.948,E2 17780.948} C_VEL
LIN {X 0,Y 391.992,Z 360.972,A -85,B 0,C 180,E1 17780.19,E2 17780.19} C_VEL
LIN {X 0,Y 406.263,Z 353.979,A -85,B 0,C 180,E1 17778,E2 17778} C_VEL
LIN {X 0,Y 407.01,Z 355.597,A -85,B 0,C 180,E1 17777.644,E2 17777.644} C_VEL
LIN {X 0,Y 409.691,Z 359.413,A -85,B 0,C 180,E1 17777.123,E2 17777.123} C_VEL
LIN {X 0,Y 406.402,Z 429.003,A -85,B 0,C 180,E1 17775.762,E2 17775.762} C_VEL
LIN {X 0,Y 402.123,Z 491.683,A -85,B 0,C 180,E1 17774.323,E2 17774.323} C_VEL
LIN {X 0,Y 396.272,Z 561.04,A -85,B 0,C 180,E1 17772.469,E2 17772.469} C_VEL
LIN {X 0,Y 393.451,Z 595.047,A -85,B 0,C 180,E1 17771.382,E2 17771.382} C_VEL
LIN {X 0,Y 391.265,Z 615.894,A -85,B 0,C 180,E1 17770.42,E2 17770.42} C_VEL
LIN {X 0,Y 388.665,Z 635.216,A -85,B 0,C 180,E1 17769.254,E2 17769.254} C_VEL
LIN {X 0,Y 385.622,Z 654.06,A -85,B 0,C 180,E1 17767.822,E2 17767.822} C_VEL
LIN {X 0,Y 382.341,Z 671.855,A -85,B 0,C 180,E1 17766.159,E2 17766.159} C_VEL
LIN {X 0,Y 379.031,Z 688.166,A -85,B 0,C 180,E1 17764.319,E2 17764.319} C_VEL
LIN {X 0,Y 376.914,Z 694.198,A -85,B 0,C 180,E1 17763.649,E2 17763.649} C_VEL
LIN {X 0,Y 368.473,Z 709.174,A -85,B 0,C 180,E1 17762.041,E2 17762.041} C_VEL
LIN {X 0,Y 366.325,Z 714.557,A -85,B 0,C 180,E1 17761.239,E2 17761.239} C_VEL
LIN {X 0,Y 363.153,Z 727.741,A -85,B 0,C 180,E1 17758.805,E2 17758.805} C_VEL
LIN {X 0,Y 360.133,Z 740.324,A -85,B 0,C 180,E1 17756.019,E2 17756.019} C_VEL
LIN {X 0,Y 357.591,Z 751.407,A -85,B 0,C 180,E1 17753.045,E2 17753.045} C_VEL
LIN {X 0,Y 355.658,Z 760.529,A -85,B 0,C 180,E1 17750.059,E2 17750.059} C_VEL
LIN {X 0,Y 354.145,Z 768.593,A -85,B 0,C 180,E1 17746.737,E2 17746.737} C_VEL
LIN {X 0,Y 353.209,Z 774.74,A -85,B 0,C 180,E1 17743.422,E2 17743.422} C_VEL
LIN {X 0,Y 352.686,Z 779.096,A -85,B 0,C 180,E1 17740.124,E2 17740.124} C_VEL
LIN {X 0,Y 352.448,Z 781.751,A -85,B 0,C 180,E1 17736.818,E2 17736.818} C_VEL
LIN {X 0,Y 352.365,Z 782.727,A -85,B 0,C 180,E1 17733.742,E2 17733.742} C_VEL
LIN {X 0,Y 352.376,Z 782.221,A -85,B 0,C 180,E1 17730.488,E2 17730.488} C_VEL
LIN {X 0,Y 352.518,Z 780.116,A -85,B 0,C 180,E1 17727.236,E2 17727.236} C_VEL
LIN {X 0,Y 352.864,Z 776.467,A -85,B 0,C 180,E1 17724.037,E2 17724.037} C_VEL
LIN {X 0,Y 353.505,Z 771.288,A -85,B 0,C 180,E1 17720.886,E2 17720.886} C_VEL
LIN {X 0,Y 354.631,Z 764.128,A -85,B 0,C 180,E1 17717.627,E2 17717.627} C_VEL
LIN {X 0,Y 356.328,Z 754.975,A -85,B 0,C 180,E1 17714.373,E2 17714.373} C_VEL
LIN {X 0,Y 358.556,Z 744.213,A -85,B 0,C 180,E1 17711.296,E2 17711.296} C_VEL
LIN {X 0,Y 361.243,Z 732.025,A -85,B 0,C 180,E1 17708.435,E2 17708.435} C_VEL
LIN {X 0,Y 364.221,Z 718.823,A -85,B 0,C 180,E1 17705.856,E2 17705.856} C_VEL
LIN {X 0,Y 367.561,Z 703.856,A -85,B 0,C 180,E1 17703.418,E2 17703.418} C_VEL
LIN {X 0,Y 370.993,Z 687.848,A -85,B 0,C 180,E1 17701.244,E2 17701.244} C_VEL
LIN {X 0,Y 374.418,Z 670.629,A -85,B 0,C 180,E1 17699.304,E2 17699.304} C_VEL
LIN {X 0,Y 377.706,Z 652.369,A -85,B 0,C 180,E1 17697.615,E2 17697.615} C_VEL
LIN {X 0,Y 380.577,Z 634.185,A -85,B 0,C 180,E1 17696.244,E2 17696.244} C_VEL
LIN {X 0,Y 383.157,Z 614.315,A -85,B 0,C 180,E1 17695.055,E2 17695.055} C_VEL
LIN {X 0,Y 385.217,Z 593.916,A -85,B 0,C 180,E1 17694.13,E2 17694.13} C_VEL
LIN {X 0,Y 388.451,Z 555.028,A -85,B 0,C 180,E1 17692.895,E2 17692.895} C_VEL
LIN {X 0,Y 394.043,Z 487.657,A -85,B 0,C 180,E1 17691.084,E2 17691.084} C_VEL
LIN {X 0,Y 398.24,Z 424.622,A -85,B 0,C 180,E1 17689.639,E2 17689.639} C_VEL
LIN {X 0,Y 401.202,Z 357.158,A -85,B 0,C 180,E1 17688.299,E2 17688.299} C_VEL
LIN {X 0,Y 399.026,Z 354.033,A -85,B 0,C 180,E1 17687.877,E2 17687.877} C_VEL
LIN {X 0,Y 393.127,Z 339.922,A -85,B 0,C 180,E1 17684.586,E2 17684.586} C_VEL
LIN {X 0,Y 387.621,Z 327.867,A -85,B 0,C 180,E1 17681.327,E2 17681.327} C_VEL
LIN {X 0,Y 383.011,Z 318.554,A -85,B 0,C 180,E1 17678.412,E2 17678.412} C_VEL
LIN {X 0,Y 379.981,Z 312.702,A -85,B 0,C 180,E1 17676.355,E2 17676.355} C_VEL
LIN {X 0,Y 372.891,Z 315.167,A -85,B 0,C 180,E1 17674.456,E2 17674.456} C_VEL
LIN {X 0,Y 370.884,Z 315.823,A -85,B 0,C 180,E1 17673.867,E2 17673.867} C_VEL
LIN {X 0,Y 370.597,Z 315.823,A -85,B 0,C 180,E1 17673.719,E2 17673.719} C_VEL
LIN {X 0,Y 371.12,Z 318.344,A -85,B 0,C 180,E1 17673.424,E2 17673.424} C_VEL
LIN {X 0,Y 369.115,Z 360.487,A -85,B 0,C 180,E1 17669.45,E2 17669.45} C_VEL
LIN {X 0,Y 366.943,Z 404.546,A -85,B 0,C 180,E1 17665.329,E2 17665.329} C_VEL
LIN {X 0,Y 364.76,Z 449.746,A -85,B 0,C 180,E1 17661.129,E2 17661.129} C_VEL
LIN {X 0,Y 363.962,Z 462.959,A -85,B 0,C 180,E1 17659.943,E2 17659.943} C_VEL
LIN {X 0,Y 360.168,Z 603.26,A -85,B 0,C 180,E1 17656.475,E2 17656.475} C_VEL
LIN {X 0,Y 359.917,Z 620.33,A -85,B 0,C 180,E1 17655.85,E2 17655.85} C_VEL
LIN {X 0,Y 359.41,Z 637.055,A -85,B 0,C 180,E1 17654.941,E2 17654.941} C_VEL
LIN {X 0,Y 358.684,Z 653.612,A -85,B 0,C 180,E1 17653.707,E2 17653.707} C_VEL
LIN {X 0,Y 357.933,Z 667.8,A -85,B 0,C 180,E1 17652.34,E2 17652.34} C_VEL
LIN {X 0,Y 357.07,Z 682.017,A -85,B 0,C 180,E1 17650.62,E2 17650.62} C_VEL
LIN {X 0,Y 356.246,Z 694.505,A -85,B 0,C 180,E1 17648.718,E2 17648.718} C_VEL
LIN {X 0,Y 355.585,Z 704.753,A -85,B 0,C 180,E1 17646.783,E2 17646.783} C_VEL
LIN {X 0,Y 355.03,Z 714.305,A -85,B 0,C 180,E1 17644.523,E2 17644.523} C_VEL
LIN {X 0,Y 354.67,Z 721.667,A -85,B 0,C 180,E1 17642.263,E2 17642.263} C_VEL
LIN {X 0,Y 354.485,Z 727.603,A -85,B 0,C 180,E1 17639.839,E2 17639.839} C_VEL
LIN {X 0,Y 354.479,Z 731.832,A -85,B 0,C 180,E1 17637.252,E2 17637.252} C_VEL
LIN {X 0,Y 354.647,Z 733.957,A -85,B 0,C 180,E1 17634.824,E2 17634.824} C_VEL
LIN {X 0,Y 354.976,Z 734.357,A -85,B 0,C 180,E1 17632.393,E2 17632.393} C_VEL
LIN {X 0,Y 355.48,Z 732.92,A -85,B 0,C 180,E1 17629.958,E2 17629.958} C_VEL
LIN {X 0,Y 356.185,Z 729.654,A -85,B 0,C 180,E1 17627.518,E2 17627.518} C_VEL
LIN {X 0,Y 357.019,Z 724.693,A -85,B 0,C 180,E1 17625.236,E2 17625.236} C_VEL
LIN {X 0,Y 358.002,Z 718.338,A -85,B 0,C 180,E1 17623.115,E2 17623.115} C_VEL
LIN {X 0,Y 359.051,Z 710.562,A -85,B 0,C 180,E1 17621.154,E2 17621.154} C_VEL
LIN {X 0,Y 360.262,Z 700.67,A -85,B 0,C 180,E1 17619.192,E2 17619.192} C_VEL
LIN {X 0,Y 361.459,Z 689.003,A -85,B 0,C 180,E1 17617.388,E2 17617.388} C_VEL
LIN {X 0,Y 362.538,Z 676.302,A -85,B 0,C 180,E1 17615.835,E2 17615.835} C_VEL
LIN {X 0,Y 363.488,Z 661.962,A -85,B 0,C 180,E1 17614.455,E2 17614.455} C_VEL
LIN {X 0,Y 364.228,Z 645.928,A -85,B 0,C 180,E1 17613.288,E2 17613.288} C_VEL
LIN {X 0,Y 364.681,Z 628.583,A -85,B 0,C 180,E1 17612.373,E2 17612.373} C_VEL
LIN {X 0,Y 364.93,Z 604.625,A -85,B 0,C 180,E1 17611.558,E2 17611.558} C_VEL
LIN {X 0,Y 368.176,Z 542.184,A -85,B 0,C 180,E1 17609.678,E2 17609.678} C_VEL
LIN {X 0,Y 372.099,Z 487.196,A -85,B 0,C 180,E1 17607.948,E2 17607.948} C_VEL
LIN {X 0,Y 375.892,Z 471.082,A -85,B 0,C 180,E1 17606.874,E2 17606.874} C_VEL
LIN {X 0,Y 376.893,Z 459.478,A -85,B 0,C 180,E1 17605.778,E2 17605.778} C_VEL
LIN {X 0,Y 379.197,Z 459.154,A -85,B 0,C 180,E1 17605.466,E2 17605.466} C_VEL
LIN {X 0,Y 383.007,Z 457.044,A -85,B 0,C 180,E1 17605.131,E2 17605.131} C_VEL
LIN {X 0,Y 387.351,Z 455.421,A -85,B 0,C 180,E1 17604.676,E2 17604.676} C_VEL
LIN {X 0,Y 390.169,Z 453.978,A -85,B 0,C 180,E1 17604.429,E2 17604.429} C_VEL
LIN {X 0,Y 406.615,Z 447.164,A -85,B 0,C 180,E1 17602.911,E2 17602.911} C_VEL
LIN {X 0,Y 412.001,Z 463.383,A -85,B 0,C 180,E1 17600.699,E2 17600.699} C_VEL
LIN {X 0,Y 419.917,Z 479.283,A -85,B 0,C 180,E1 17598.37,E2 17598.37} C_VEL
LIN {X 0,Y 422.808,Z 483.968,A -85,B 0,C 180,E1 17597.657,E2 17597.657} C_VEL
LIN {X 0,Y 415.833,Z 497.666,A -85,B 0,C 180,E1 17597.17,E2 17597.17} C_VEL
LIN {X 0,Y 406.146,Z 516.656,A -85,B 0,C 180,E1 17596.47,E2 17596.47} C_VEL
LIN {X 0,Y 401.969,Z 526.44,A -85,B 0,C 180,E1 17596.063,E2 17596.063} C_VEL
LIN {X 0,Y 398.05,Z 553.446,A -85,B 0,C 180,E1 17595.923,E2 17595.923} C_VEL
LIN {X 0,Y 395.958,Z 574.16,A -85,B 0,C 180,E1 17595.618,E2 17595.618} C_VEL
LIN {X 0,Y 393.599,Z 601.318,A -85,B 0,C 180,E1 17594.871,E2 17594.871} C_VEL
LIN {X 0,Y 390.121,Z 629.096,A -85,B 0,C 180,E1 17593.865,E2 17593.865} C_VEL
LIN {X 0,Y 386.573,Z 653.948,A -85,B 0,C 180,E1 17592.661,E2 17592.661} C_VEL
LIN {X 0,Y 382.718,Z 678.355,A -85,B 0,C 180,E1 17591.175,E2 17591.175} C_VEL
LIN {X 0,Y 378.912,Z 700.88,A -85,B 0,C 180,E1 17589.49,E2 17589.49} C_VEL
LIN {X 0,Y 375.118,Z 721.668,A -85,B 0,C 180,E1 17587.618,E2 17587.618} C_VEL
LIN {X 0,Y 371.528,Z 739.927,A -85,B 0,C 180,E1 17585.636,E2 17585.636} C_VEL
LIN {X 0,Y 368.019,Z 756.411,A -85,B 0,C 180,E1 17583.472,E2 17583.472} C_VEL
LIN {X 0,Y 364.441,Z 772.492,A -85,B 0,C 180,E1 17580.958,E2 17580.958} C_VEL
LIN {X 0,Y 361.203,Z 786.863,A -85,B 0,C 180,E1 17578.252,E2 17578.252} C_VEL
LIN {X 0,Y 358.345,Z 799.981,A -85,B 0,C 180,E1 17575.308,E2 17575.308} C_VEL
LIN {X 0,Y 355.845,Z 812.285,A -85,B 0,C 180,E1 17571.944,E2 17571.944} C_VEL
LIN {X 0,Y 354.175,Z 821.771,A -85,B 0,C 180,E1 17568.774,E2 17568.774} C_VEL
LIN {X 0,Y 352.984,Z 830.219,A -85,B 0,C 180,E1 17565.274,E2 17565.274} C_VEL
LIN {X 0,Y 352.37,Z 836.706,A -85,B 0,C 180,E1 17561.78,E2 17561.78} C_VEL
LIN {X 0,Y 352.15,Z 841.44,A -85,B 0,C 180,E1 17558.326,E2 17558.326} C_VEL
LIN {X 0,Y 352.144,Z 844.455,A -85,B 0,C 180,E1 17554.886,E2 17554.886} C_VEL
LIN {X 0,Y 352.179,Z 845.875,A -85,B 0,C 180,E1 17551.627,E2 17551.627} C_VEL
LIN {X 0,Y 352.179,Z 845.873,A -85,B 0,C 180,E1 17548.373,E2 17548.373} C_VEL
LIN {X 0,Y 352.145,Z 844.444,A -85,B 0,C 180,E1 17545.114,E2 17545.114} C_VEL
LIN {X 0,Y 352.15,Z 841.429,A -85,B 0,C 180,E1 17541.674,E2 17541.674} C_VEL
LIN {X 0,Y 352.369,Z 836.714,A -85,B 0,C 180,E1 17538.211,E2 17538.211} C_VEL
LIN {X 0,Y 352.983,Z 830.301,A -85,B 0,C 180,E1 17534.726,E2 17534.726} C_VEL
LIN {X 0,Y 354.174,Z 821.936,A -85,B 0,C 180,E1 17531.226,E2 17531.226} C_VEL
LIN {X 0,Y 355.961,Z 812.046,A -85,B 0,C 180,E1 17527.889,E2 17527.889} C_VEL
LIN {X 0,Y 358.49,Z 799.952,A -85,B 0,C 180,E1 17524.563,E2 17524.563} C_VEL
LIN {X 0,Y 361.449,Z 786.853,A -85,B 0,C 180,E1 17521.589,E2 17521.589} C_VEL
LIN {X 0,Y 364.974,Z 771.75,A -85,B 0,C 180,E1 17518.729,E2 17518.729} C_VEL
LIN {X 0,Y 368.809,Z 755.202,A -85,B 0,C 180,E1 17516.143,E2 17516.143} C_VEL
LIN {X 0,Y 372.449,Z 738.734,A -85,B 0,C 180,E1 17513.99,E2 17513.99} C_VEL
LIN {X 0,Y 376.325,Z 719.792,A -85,B 0,C 180,E1 17511.946,E2 17511.946} C_VEL
LIN {X 0,Y 380.396,Z 698.034,A -85,B 0,C 180,E1 17510.018,E2 17510.018} C_VEL
LIN {X 0,Y 384.414,Z 675.347,A -85,B 0,C 180,E1 17508.351,E2 17508.351} C_VEL
LIN {X 0,Y 388.211,Z 652.201,A -85,B 0,C 180,E1 17506.958,E2 17506.958} C_VEL
LIN {X 0,Y 392.076,Z 626.273,A -85,B 0,C 180,E1 17505.729,E2 17505.729} C_VEL
LIN {X 0,Y 395.454,Z 600.122,A -85,B 0,C 180,E1 17504.797,E2 17504.797} C_VEL
LIN {X 0,Y 397.955,Z 573.033,A -85,B 0,C 180,E1 17504.063,E2 17504.063} C_VEL
LIN {X 0,Y 400.255,Z 553.493,A -85,B 0,C 180,E1 17503.81,E2 17503.81} C_VEL
LIN {X 0,Y 403.464,Z 533.066,A -85,B 0,C 180,E1 17503.754,E2 17503.754} C_VEL
LIN {X 0,Y 404.789,Z 525.285,A -85,B 0,C 180,E1 17503.738,E2 17503.738} C_VEL
LIN {X 0,Y 412.634,Z 511.153,A -85,B 0,C 180,E1 17503.065,E2 17503.065} C_VEL
LIN {X 0,Y 405.494,Z 497.305,A -85,B 0,C 180,E1 17500.799,E2 17500.799} C_VEL
LIN {X 0,Y 400.284,Z 482.128,A -85,B 0,C 180,E1 17498.46,E2 17498.46} C_VEL
LIN {X 0,Y 397.181,Z 465.59,A -85,B 0,C 180,E1 17496.09,E2 17496.09} C_VEL
LIN {X 0,Y 396.133,Z 447.78,A -85,B 0,C 180,E1 17493.73,E2 17493.73} C_VEL
LIN {X 0,Y 397.248,Z 427.798,A -85,B 0,C 180,E1 17491.315,E2 17491.315} C_VEL
LIN {X 0,Y 398.993,Z 414.771,A -85,B 0,C 180,E1 17489.857,E2 17489.857} C_VEL
LIN {X 0,Y 389.801,Z 419.186,A -85,B 0,C 180,E1 17488.831,E2 17488.831} C_VEL
LIN {X 0,Y 383.772,Z 422.194,A -85,B 0,C 180,E1 17488.136,E2 17488.136} C_VEL
LIN {X 0,Y 379.521,Z 424.316,A -85,B 0,C 180,E1 17487.624,E2 17487.624} C_VEL
LIN {X 0,Y 377.667,Z 425.461,A -85,B 0,C 180,E1 17487.429,E2 17487.429} C_VEL
LIN {X 0,Y 374.262,Z 427.222,A -85,B 0,C 180,E1 17487.011,E2 17487.011} C_VEL
LIN {X 0,Y 372.91,Z 427.553,A -85,B 0,C 180,E1 17486.75,E2 17486.75} C_VEL
LIN {X 0,Y 370.285,Z 476.539,A -85,B 0,C 180,E1 17482.63,E2 17482.63} C_VEL
LIN {X 0,Y 368.202,Z 514.342,A -85,B 0,C 180,E1 17479.429,E2 17479.429} C_VEL
LIN {X 0,Y 365.394,Z 529.307,A -85,B 0,C 180,E1 17478.429,E2 17478.429} C_VEL
LIN {X 0,Y 361.781,Z 621.542,A -85,B 0,C 180,E1 17475.883,E2 17475.883} C_VEL
LIN {X 0,Y 361.768,Z 643.54,A -85,B 0,C 180,E1 17475.191,E2 17475.191} C_VEL
LIN {X 0,Y 361.582,Z 657.365,A -85,B 0,C 180,E1 17474.492,E2 17474.492} C_VEL
LIN {X 0,Y 361.054,Z 671.877,A -85,B 0,C 180,E1 17473.451,E2 17473.451} C_VEL
LIN {X 0,Y 360.344,Z 685.046,A -85,B 0,C 180,E1 17472.173,E2 17472.173} C_VEL
LIN {X 0,Y 359.459,Z 697.006,A -85,B 0,C 180,E1 17470.659,E2 17470.659} C_VEL
LIN {X 0,Y 358.515,Z 707.199,A -85,B 0,C 180,E1 17468.985,E2 17468.985} C_VEL
LIN {X 0,Y 357.607,Z 715.489,A -85,B 0,C 180,E1 17467.227,E2 17467.227} C_VEL
LIN {X 0,Y 356.748,Z 722.483,A -85,B 0,C 180,E1 17465.306,E2 17465.306} C_VEL
LIN {X 0,Y 355.977,Z 727.998,A -85,B 0,C 180,E1 17463.22,E2 17463.22} C_VEL
LIN {X 0,Y 355.33,Z 731.871,A -85,B 0,C 180,E1 17460.967,E2 17460.967} C_VEL
LIN {X 0,Y 354.894,Z 733.775,A -85,B 0,C 180,E1 17458.869,E2 17458.869} C_VEL
LIN {X 0,Y 354.587,Z 734.079,A -85,B 0,C 180,E1 17456.575,E2 17456.575} C_VEL
LIN {X 0,Y 354.424,Z 732.397,A -85,B 0,C 180,E1 17454.17,E2 17454.17} C_VEL
LIN {X 0,Y 354.436,Z 728.929,A -85,B 0,C 180,E1 17451.891,E2 17451.891} C_VEL
LIN {X 0,Y 354.597,Z 723.954,A -85,B 0,C 180,E1 17449.765,E2 17449.765} C_VEL
LIN {X 0,Y 354.932,Z 717.083,A -85,B 0,C 180,E1 17447.637,E2 17447.637} C_VEL
LIN {X 0,Y 355.446,Z 707.903,A -85,B 0,C 180,E1 17445.501,E2 17445.501} C_VEL
LIN {X 0,Y 356.054,Z 697.341,A -85,B 0,C 180,E1 17443.607,E2 17443.607} C_VEL
LIN {X 0,Y 356.728,Z 684.892,A -85,B 0,C 180,E1 17441.873,E2 17441.873} C_VEL
LIN {X 0,Y 357.374,Z 670.978,A -85,B 0,C 180,E1 17440.382,E2 17440.382} C_VEL
LIN {X 0,Y 357.908,Z 656.607,A -85,B 0,C 180,E1 17439.219,E2 17439.219} C_VEL
LIN {X 0,Y 358.27,Z 640.803,A -85,B 0,C 180,E1 17438.302,E2 17438.302} C_VEL
LIN {X 0,Y 358.399,Z 624.583,A -85,B 0,C 180,E1 17437.702,E2 17437.702} C_VEL
LIN {X 0,Y 360.091,Z 537.593,A -85,B 0,C 180,E1 17435.603,E2 17435.603} C_VEL
LIN {X 0,Y 360.803,Z 512.746,A -85,B 0,C 180,E1 17434.985,E2 17434.985} C_VEL
LIN {X 0,Y 361.911,Z 503.744,A -85,B 0,C 180,E1 17434.244,E2 17434.244} C_VEL
LIN {X 0,Y 364.139,Z 453.1,A -85,B 0,C 180,E1 17429.835,E2 17429.835} C_VEL
LIN {X 0,Y 366.347,Z 405.938,A -85,B 0,C 180,E1 17425.709,E2 17425.709} C_VEL
LIN {X 0,Y 367.251,Z 388.923,A -85,B 0,C 180,E1 17424.186,E2 17424.186} C_VEL
LIN {X 0,Y 368.383,Z 389.492,A -85,B 0,C 180,E1 17423.915,E2 17423.915} C_VEL
LIN {X 0,Y 370.691,Z 388.007,A -85,B 0,C 180,E1 17423.456,E2 17423.456} C_VEL
LIN {X 0,Y 374.228,Z 383.184,A -85,B 0,C 180,E1 17422.855,E2 17422.855} C_VEL
LIN {X 0,Y 377.119,Z 377.772,A -85,B 0,C 180,E1 17422.424,E2 17422.424} C_VEL
LIN {X 0,Y 380.457,Z 375.767,A -85,B 0,C 180,E1 17421.811,E2 17421.811} C_VEL
LIN {X 0,Y 382.277,Z 374.153,A -85,B 0,C 180,E1 17421.5,E2 17421.5} C_VEL
LIN {X 0,Y 386.975,Z 371.506,A -85,B 0,C 180,E1 17420.678,E2 17420.678} C_VEL
LIN {X 0,Y 403.831,Z 362.718,A -85,B 0,C 180,E1 17417.973,E2 17417.973} C_VEL
LIN {X 0,Y 404.195,Z 363.664,A -85,B 0,C 180,E1 17417.888,E2 17417.888} C_VEL
LIN {X 0,Y 400.853,Z 431.078,A -85,B 0,C 180,E1 17416.556,E2 17416.556} C_VEL
LIN {X 0,Y 396.497,Z 492.238,A -85,B 0,C 180,E1 17415.135,E2 17415.135} C_VEL
LIN {X 0,Y 390.587,Z 559.228,A -85,B 0,C 180,E1 17413.319,E2 17413.319} C_VEL
LIN {X 0,Y 387.42,Z 595.133,A -85,B 0,C 180,E1 17412.16,E2 17412.16} C_VEL
LIN {X 0,Y 385.26,Z 615.237,A -85,B 0,C 180,E1 17411.24,E2 17411.24} C_VEL
LIN {X 0,Y 382.556,Z 634.811,A -85,B 0,C 180,E1 17410.063,E2 17410.063} C_VEL
LIN {X 0,Y 379.437,Z 653.488,A -85,B 0,C 180,E1 17408.648,E2 17408.648} C_VEL
LIN {X 0,Y 375.945,Z 671.694,A -85,B 0,C 180,E1 17406.947,E2 17406.947} C_VEL
LIN {X 0,Y 372.337,Z 688.705,A -85,B 0,C 180,E1 17405.011,E2 17405.011} C_VEL
LIN {X 0,Y 368.596,Z 705.081,A -85,B 0,C 180,E1 17402.762,E2 17402.762} C_VEL
LIN {X 0,Y 366.325,Z 714.557,A -85,B 0,C 180,E1 17401.239,E2 17401.239} C_VEL
LIN {X 0,Y 364.187,Z 719.906,A -85,B 0,C 180,E1 17400.402,E2 17400.402} C_VEL
LIN {X 0,Y 355.711,Z 732.895,A -85,B 0,C 180,E1 17398.369,E2 17398.369} C_VEL
LIN {X 0,Y 353.671,Z 737.462,A -85,B 0,C 180,E1 17397.421,E2 17397.421} C_VEL
LIN {X 0,Y 350.773,Z 749.1,A -85,B 0,C 180,E1 17394.414,E2 17394.414} C_VEL
LIN {X 0,Y 348.411,Z 759.227,A -85,B 0,C 180,E1 17391.198,E2 17391.198} C_VEL
LIN {X 0,Y 346.668,Z 767.604,A -85,B 0,C 180,E1 17387.862,E2 17387.862} C_VEL
LIN {X 0,Y 345.535,Z 773.98,A -85,B 0,C 180,E1 17384.581,E2 17384.581} C_VEL
LIN {X 0,Y 344.872,Z 778.789,A -85,B 0,C 180,E1 17381.201,E2 17381.201} C_VEL
LIN {X 0,Y 344.533,Z 781.889,A -85,B 0,C 180,E1 17377.84,E2 17377.84} C_VEL
LIN {X 0,Y 344.411,Z 783.336,A -85,B 0,C 180,E1 17374.663,E2 17374.663} C_VEL
LIN {X 0,Y 344.403,Z 783.279,A -85,B 0,C 180,E1 17371.331,E2 17371.331} C_VEL
LIN {X 0,Y 344.511,Z 781.573,A -85,B 0,C 180,E1 17368.004,E2 17368.004} C_VEL
LIN {X 0,Y 344.792,Z 778.446,A -85,B 0,C 180,E1 17364.842,E2 17364.842} C_VEL
LIN {X 0,Y 345.399,Z 773.544,A -85,B 0,C 180,E1 17361.51,E2 17361.51} C_VEL
LIN {X 0,Y 346.467,Z 766.869,A -85,B 0,C 180,E1 17358.177,E2 17358.177} C_VEL
LIN {X 0,Y 348.012,Z 758.748,A -85,B 0,C 180,E1 17355.014,E2 17355.014} C_VEL
LIN {X 0,Y 350.171,Z 748.693,A -85,B 0,C 180,E1 17351.866,E2 17351.866} C_VEL
LIN {X 0,Y 352.829,Z 737.127,A -85,B 0,C 180,E1 17348.906,E2 17348.906} C_VEL
LIN {X 0,Y 355.934,Z 724.056,A -85,B 0,C 180,E1 17346.139,E2 17346.139} C_VEL
LIN {X 0,Y 359.388,Z 709.437,A -85,B 0,C 180,E1 17343.568,E2 17343.568} C_VEL
LIN {X 0,Y 362.98,Z 693.728,A -85,B 0,C 180,E1 17341.27,E2 17341.27} C_VEL
LIN {X 0,Y 366.61,Z 676.811,A -85,B 0,C 180,E1 17339.217,E2 17339.217} C_VEL
LIN {X 0,Y 370.01,Z 659.367,A -85,B 0,C 180,E1 17337.469,E2 17337.469} C_VEL
LIN {X 0,Y 373.194,Z 640.788,A -85,B 0,C 180,E1 17335.947,E2 17335.947} C_VEL
LIN {X 0,Y 376.048,Z 621.193,A -85,B 0,C 180,E1 17334.669,E2 17334.669} C_VEL
LIN {X 0,Y 378.361,Z 600.985,A -85,B 0,C 180,E1 17333.652,E2 17333.652} C_VEL
LIN {X 0,Y 380.606,Z 575.238,A -85,B 0,C 180,E1 17332.721,E2 17332.721} C_VEL
LIN {X 0,Y 386.621,Z 508.179,A -85,B 0,C 180,E1 17330.799,E2 17330.799} C_VEL
LIN {X 0,Y 391.233,Z 446.829,A -85,B 0,C 180,E1 17329.294,E2 17329.294} C_VEL
LIN {X 0,Y 394.439,Z 388.727,A -85,B 0,C 180,E1 17328.082,E2 17328.082} C_VEL
LIN {X 0,Y 395.49,Z 360.978,A -85,B 0,C 180,E1 17327.527,E2 17327.527} C_VEL
LIN {X 0,Y 392.576,Z 356.834,A -85,B 0,C 180,E1 17326.955,E2 17326.955} C_VEL
LIN {X 0,Y 387.125,Z 343.884,A -85,B 0,C 180,E1 17323.804,E2 17323.804} C_VEL
LIN {X 0,Y 382.316,Z 333.171,A -85,B 0,C 180,E1 17320.831,E2 17320.831} C_VEL
LIN {X 0,Y 377.202,Z 322.364,A -85,B 0,C 180,E1 17317.375,E2 17317.375} C_VEL
LIN {X 0,Y 375.653,Z 319.982,A -85,B 0,C 180,E1 17316.41,E2 17316.41} C_VEL
LIN {X 0,Y 367.889,Z 322.848,A -85,B 0,C 180,E1 17314.33,E2 17314.33} C_VEL
LIN {X 0,Y 365.071,Z 325.081,A -85,B 0,C 180,E1 17313.779,E2 17313.779} C_VEL
LIN {X 0,Y 363.611,Z 325.81,A -85,B 0,C 180,E1 17313.342,E2 17313.342} C_VEL
LIN {X 0,Y 361.492,Z 368.221,A -85,B 0,C 180,E1 17309.313,E2 17309.313} C_VEL
LIN {X 0,Y 359.237,Z 411.74,A -85,B 0,C 180,E1 17305.205,E2 17305.205} C_VEL
LIN {X 0,Y 356.955,Z 457.361,A -85,B 0,C 180,E1 17300.925,E2 17300.925} C_VEL
LIN {X 0,Y 356.398,Z 464.067,A -85,B 0,C 180,E1 17300.347,E2 17300.347} C_VEL
LIN {X 0,Y 352.433,Z 603.208,A -85,B 0,C 180,E1 17296.807,E2 17296.807} C_VEL
LIN {X 0,Y 352.176,Z 620.827,A -85,B 0,C 180,E1 17296.166,E2 17296.166} C_VEL
LIN {X 0,Y 351.632,Z 638.131,A -85,B 0,C 180,E1 17295.209,E2 17295.209} C_VEL
LIN {X 0,Y 350.918,Z 653.912,A -85,B 0,C 180,E1 17294.016,E2 17294.016} C_VEL
LIN {X 0,Y 350.138,Z 668.341,A -85,B 0,C 180,E1 17292.619,E2 17292.619} C_VEL
LIN {X 0,Y 349.255,Z 682.491,A -85,B 0,C 180,E1 17290.892,E2 17290.892} C_VEL
LIN {X 0,Y 348.449,Z 694.368,A -85,B 0,C 180,E1 17289.081,E2 17289.081} C_VEL
LIN {X 0,Y 347.753,Z 704.969,A -85,B 0,C 180,E1 17287.102,E2 17287.102} C_VEL
LIN {X 0,Y 347.153,Z 714.874,A -85,B 0,C 180,E1 17284.763,E2 17284.763} C_VEL
LIN {X 0,Y 346.781,Z 722.415,A -85,B 0,C 180,E1 17282.479,E2 17282.479} C_VEL
LIN {X 0,Y 346.586,Z 728.583,A -85,B 0,C 180,E1 17280.001,E2 17280.001} C_VEL
LIN {X 0,Y 346.571,Z 732.786,A -85,B 0,C 180,E1 17277.52,E2 17277.52} C_VEL
LIN {X 0,Y 346.753,Z 735.254,A -85,B 0,C 180,E1 17275.038,E2 17275.038} C_VEL
LIN {X 0,Y 347.088,Z 735.897,A -85,B 0,C 180,E1 17272.552,E2 17272.552} C_VEL
LIN {X 0,Y 347.631,Z 734.792,A -85,B 0,C 180,E1 17270.063,E2 17270.063} C_VEL
LIN {X 0,Y 348.373,Z 731.769,A -85,B 0,C 180,E1 17267.57,E2 17267.57} C_VEL
LIN {X 0,Y 349.273,Z 727.165,A -85,B 0,C 180,E1 17265.24,E2 17265.24} C_VEL
LIN {X 0,Y 350.391,Z 720.499,A -85,B 0,C 180,E1 17262.908,E2 17262.908} C_VEL
LIN {X 0,Y 351.54,Z 712.963,A -85,B 0,C 180,E1 17260.909,E2 17260.909} C_VEL
LIN {X 0,Y 352.828,Z 703.217,A -85,B 0,C 180,E1 17258.907,E2 17258.907} C_VEL
LIN {X 0,Y 354.13,Z 691.869,A -85,B 0,C 180,E1 17257.069,E2 17257.069} C_VEL
LIN {X 0,Y 355.312,Z 679.435,A -85,B 0,C 180,E1 17255.477,E2 17255.477} C_VEL
LIN {X 0,Y 356.428,Z 664.273,A -85,B 0,C 180,E1 17253.959,E2 17253.959} C_VEL
LIN {X 0,Y 357.256,Z 648.529,A -85,B 0,C 180,E1 17252.769,E2 17252.769} C_VEL
LIN {X 0,Y 357.802,Z 630.544,A -85,B 0,C 180,E1 17251.782,E2 17251.782} C_VEL
LIN {X 0,Y 358.161,Z 606.558,A -85,B 0,C 180,E1 17250.922,E2 17250.922} C_VEL
LIN {X 0,Y 361.402,Z 549.752,A -85,B 0,C 180,E1 17249.129,E2 17249.129} C_VEL
LIN {X 0,Y 366.093,Z 489.85,A -85,B 0,C 180,E1 17247.171,E2 17247.171} C_VEL
LIN {X 0,Y 370.096,Z 473.222,A -85,B 0,C 180,E1 17246.091,E2 17246.091} C_VEL
LIN {X 0,Y 370.583,Z 469.028,A -85,B 0,C 180,E1 17245.675,E2 17245.675} C_VEL
LIN {X 0,Y 373.269,Z 468.531,A -85,B 0,C 180,E1 17245.321,E2 17245.321} C_VEL
LIN {X 0,Y 377.617,Z 466.18,A -85,B 0,C 180,E1 17244.931,E2 17244.931} C_VEL
LIN {X 0,Y 382.116,Z 464.233,A -85,B 0,C 180,E1 17244.487,E2 17244.487} C_VEL
LIN {X 0,Y 397.632,Z 457.415,A -85,B 0,C 180,E1 17243.061,E2 17243.061} C_VEL
LIN {X 0,Y 401.544,Z 455.716,A -85,B 0,C 180,E1 17242.721,E2 17242.721} C_VEL
LIN {X 0,Y 407.642,Z 472.244,A -85,B 0,C 180,E1 17240.378,E2 17240.378} C_VEL
LIN {X 0,Y 415.034,Z 486.479,A -85,B 0,C 180,E1 17238.247,E2 17238.247} C_VEL
LIN {X 0,Y 409.234,Z 497.614,A -85,B 0,C 180,E1 17237.862,E2 17237.862} C_VEL
LIN {X 0,Y 399.587,Z 516.638,A -85,B 0,C 180,E1 17237.152,E2 17237.152} C_VEL
LIN {X 0,Y 396.418,Z 524.053,A -85,B 0,C 180,E1 17236.85,E2 17236.85} C_VEL
LIN {X 0,Y 392.237,Z 552.487,A -85,B 0,C 180,E1 17236.714,E2 17236.714} C_VEL
LIN {X 0,Y 389.971,Z 573.976,A -85,B 0,C 180,E1 17236.394,E2 17236.394} C_VEL
LIN {X 0,Y 387.321,Z 602.264,A -85,B 0,C 180,E1 17235.59,E2 17235.59} C_VEL
LIN {X 0,Y 383.866,Z 628.658,A -85,B 0,C 180,E1 17234.614,E2 17234.614} C_VEL
LIN {X 0,Y 380.073,Z 654.077,A -85,B 0,C 180,E1 17233.363,E2 17233.363} C_VEL
LIN {X 0,Y 376.085,Z 678.422,A -85,B 0,C 180,E1 17231.86,E2 17231.86} C_VEL
LIN {X 0,Y 372.116,Z 700.784,A -85,B 0,C 180,E1 17230.156,E2 17230.156} C_VEL
LIN {X 0,Y 367.867,Z 723.222,A -85,B 0,C 180,E1 17228.097,E2 17228.097} C_VEL
LIN {X 0,Y 364.287,Z 740.437,A -85,B 0,C 180,E1 17226.165,E2 17226.165} C_VEL
LIN {X 0,Y 360.386,Z 757.945,A -85,B 0,C 180,E1 17223.798,E2 17223.798} C_VEL
LIN {X 0,Y 356.913,Z 772.713,A -85,B 0,C 180,E1 17221.404,E2 17221.404} C_VEL
LIN {X 0,Y 353.456,Z 787.42,A -85,B 0,C 180,E1 17218.56,E2 17218.56} C_VEL
LIN {X 0,Y 350.615,Z 799.789,A -85,B 0,C 180,E1 17215.688,E2 17215.688} C_VEL
LIN {X 0,Y 348.025,Z 811.948,A -85,B 0,C 180,E1 17212.286,E2 17212.286} C_VEL
LIN {X 0,Y 346.199,Z 821.806,A -85,B 0,C 180,E1 17208.873,E2 17208.873} C_VEL
LIN {X 0,Y 345.029,Z 829.769,A -85,B 0,C 180,E1 17205.463,E2 17205.463} C_VEL
LIN {X 0,Y 344.37,Z 836.455,A -85,B 0,C 180,E1 17201.727,E2 17201.727} C_VEL
LIN {X 0,Y 344.167,Z 840.865,A -85,B 0,C 180,E1 17198.352,E2 17198.352} C_VEL
LIN {X 0,Y 344.172,Z 843.831,A -85,B 0,C 180,E1 17194.833,E2 17194.833} C_VEL
LIN {X 0,Y 344.212,Z 845.198,A -85,B 0,C 180,E1 17191.498,E2 17191.498} C_VEL
LIN {X 0,Y 344.209,Z 845.116,A -85,B 0,C 180,E1 17188.169,E2 17188.169} C_VEL
LIN {X 0,Y 344.164,Z 843.518,A -85,B 0,C 180,E1 17184.666,E2 17184.666} C_VEL
LIN {X 0,Y 344.166,Z 840.536,A -85,B 0,C 180,E1 17181.311,E2 17181.311} C_VEL
LIN {X 0,Y 344.424,Z 835.731,A -85,B 0,C 180,E1 17177.765,E2 17177.765} C_VEL
LIN {X 0,Y 345.119,Z 829.221,A -85,B 0,C 180,E1 17174.197,E2 17174.197} C_VEL
LIN {X 0,Y 346.424,Z 820.742,A -85,B 0,C 180,E1 17170.615,E2 17170.615} C_VEL
LIN {X 0,Y 348.268,Z 811.289,A -85,B 0,C 180,E1 17167.374,E2 17167.374} C_VEL
LIN {X 0,Y 350.96,Z 799.143,A -85,B 0,C 180,E1 17163.976,E2 17163.976} C_VEL
LIN {X 0,Y 353.913,Z 786.821,A -85,B 0,C 180,E1 17161.112,E2 17161.112} C_VEL
LIN {X 0,Y 357.581,Z 771.87,A -85,B 0,C 180,E1 17158.215,E2 17158.215} C_VEL
LIN {X 0,Y 361.351,Z 756.484,A -85,B 0,C 180,E1 17155.73,E2 17155.73} C_VEL
LIN {X 0,Y 365.419,Z 739.01,A -85,B 0,C 180,E1 17153.381,E2 17153.381} C_VEL
LIN {X 0,Y 369.306,Z 721.033,A -85,B 0,C 180,E1 17151.387,E2 17151.387} C_VEL
LIN {X 0,Y 373.765,Z 698.26,A -85,B 0,C 180,E1 17149.327,E2 17149.327} C_VEL
LIN {X 0,Y 377.876,Z 676.158,A -85,B 0,C 180,E1 17147.669,E2 17147.669} C_VEL
LIN {X 0,Y 382.014,Z 651.903,A -85,B 0,C 180,E1 17146.188,E2 17146.188} C_VEL
LIN {X 0,Y 386.099,Z 625.591,A -85,B 0,C 180,E1 17144.932,E2 17144.932} C_VEL
LIN {X 0,Y 389.646,Z 599.232,A -85,B 0,C 180,E1 17143.978,E2 17143.978} C_VEL
LIN {X 0,Y 392.319,Z 571.844,A -85,B 0,C 180,E1 17143.232,E2 17143.232} C_VEL
LIN {X 0,Y 394.869,Z 551.25,A -85,B 0,C 180,E1 17142.976,E2 17142.976} C_VEL
LIN {X 0,Y 399.504,Z 522.917,A -85,B 0,C 180,E1 17142.927,E2 17142.927} C_VEL
LIN {X 0,Y 404.746,Z 513.299,A -85,B 0,C 180,E1 17142.455,E2 17142.455} C_VEL
LIN {X 0,Y 397.449,Z 497.66,A -85,B 0,C 180,E1 17139.889,E2 17139.889} C_VEL
LIN {X 0,Y 392.763,Z 481.584,A -85,B 0,C 180,E1 17137.414,E2 17137.414} C_VEL
LIN {X 0,Y 390.264,Z 463.531,A -85,B 0,C 180,E1 17134.842,E2 17134.842} C_VEL
LIN {X 0,Y 390.036,Z 444.856,A -85,B 0,C 180,E1 17132.396,E2 17132.396} C_VEL
LIN {X 0,Y 392.068,Z 423.917,A -85,B 0,C 180,E1 17129.905,E2 17129.905} C_VEL
LIN {X 0,Y 377.677,Z 431.129,A -85,B 0,C 180,E1 17128.286,E2 17128.286} C_VEL
LIN {X 0,Y 373.282,Z 433.489,A -85,B 0,C 180,E1 17127.779,E2 17127.779} C_VEL
LIN {X 0,Y 371.59,Z 434.329,A -85,B 0,C 180,E1 17127.568,E2 17127.568} C_VEL
LIN {X 0,Y 367.994,Z 436.407,A -85,B 0,C 180,E1 17127.159,E2 17127.159} C_VEL
LIN {X 0,Y 366.281,Z 436.916,A -85,B 0,C 180,E1 17126.848,E2 17126.848} C_VEL
LIN {X 0,Y 363.177,Z 488.648,A -85,B 0,C 180,E1 17122.414,E2 17122.414} C_VEL
LIN {X 0,Y 361.631,Z 515.166,A -85,B 0,C 180,E1 17120.134,E2 17120.134} C_VEL
LIN {X 0,Y 358.557,Z 531.265,A -85,B 0,C 180,E1 17119.059,E2 17119.059} C_VEL
LIN {X 0,Y 354.694,Z 619.46,A -85,B 0,C 180,E1 17116.531,E2 17116.531} C_VEL
LIN {X 0,Y 354.555,Z 644.908,A -85,B 0,C 180,E1 17115.707,E2 17115.707} C_VEL
LIN {X 0,Y 354.317,Z 659.15,A -85,B 0,C 180,E1 17114.963,E2 17114.963} C_VEL
LIN {X 0,Y 353.75,Z 673.618,A -85,B 0,C 180,E1 17113.901,E2 17113.901} C_VEL
LIN {X 0,Y 352.978,Z 686.734,A -85,B 0,C 180,E1 17112.598,E2 17112.598} C_VEL
LIN {X 0,Y 352.014,Z 698.614,A -85,B 0,C 180,E1 17111.053,E2 17111.053} C_VEL
LIN {X 0,Y 350.997,Z 708.792,A -85,B 0,C 180,E1 17109.344,E2 17109.344} C_VEL
LIN {X 0,Y 350.022,Z 717.086,A -85,B 0,C 180,E1 17107.55,E2 17107.55} C_VEL
LIN {X 0,Y 349.084,Z 724.034,A -85,B 0,C 180,E1 17105.588,E2 17105.588} C_VEL
LIN {X 0,Y 348.242,Z 729.507,A -85,B 0,C 180,E1 17103.456,E2 17103.456} C_VEL
LIN {X 0,Y 347.537,Z 733.358,A -85,B 0,C 180,E1 17101.153,E2 17101.153} C_VEL
LIN {X 0,Y 347.057,Z 735.225,A -85,B 0,C 180,E1 17099.009,E2 17099.009} C_VEL
LIN {X 0,Y 346.718,Z 735.48,A -85,B 0,C 180,E1 17096.693,E2 17096.693} C_VEL
LIN {X 0,Y 346.531,Z 733.896,A -85,B 0,C 180,E1 17094.37,E2 17094.37} C_VEL
LIN {X 0,Y 346.522,Z 730.809,A -85,B 0,C 180,E1 17092.205,E2 17092.205} C_VEL
LIN {X 0,Y 346.672,Z 725.597,A -85,B 0,C 180,E1 17089.866,E2 17089.866} C_VEL
LIN {X 0,Y 347.014,Z 718.551,A -85,B 0,C 180,E1 17087.628,E2 17087.628} C_VEL
LIN {X 0,Y 347.518,Z 709.652,A -85,B 0,C 180,E1 17085.503,E2 17085.503} C_VEL
LIN {X 0,Y 348.166,Z 698.647,A -85,B 0,C 180,E1 17083.482,E2 17083.482} C_VEL
LIN {X 0,Y 348.862,Z 686.179,A -85,B 0,C 180,E1 17081.709,E2 17081.709} C_VEL
LIN {X 0,Y 349.531,Z 672.349,A -85,B 0,C 180,E1 17080.193,E2 17080.193} C_VEL
LIN {X 0,Y 350.085,Z 657.903,A -85,B 0,C 180,E1 17078.995,E2 17078.995} C_VEL
LIN {X 0,Y 350.473,Z 642.066,A -85,B 0,C 180,E1 17078.054,E2 17078.054} C_VEL
LIN {X 0,Y 350.613,Z 625.72,A -85,B 0,C 180,E1 17077.431,E2 17077.431} C_VEL
LIN {X 0,Y 352.279,Z 542.614,A -85,B 0,C 180,E1 17075.363,E2 17075.363} C_VEL
LIN {X 0,Y 353.181,Z 513.473,A -85,B 0,C 180,E1 17074.602,E2 17074.602} C_VEL
LIN {X 0,Y 354.352,Z 503.948,A -85,B 0,C 180,E1 17073.805,E2 17073.805} C_VEL
LIN {X 0,Y 356.656,Z 453.758,A -85,B 0,C 180,E1 17069.391,E2 17069.391} C_VEL
LIN {X 0,Y 358.906,Z 409.34,A -85,B 0,C 180,E1 17065.433,E2 17065.433} C_VEL
LIN {X 0,Y 360.158,Z 409.801,A -85,B 0,C 180,E1 17065.117,E2 17065.117} C_VEL
LIN {X 0,Y 362.431,Z 408.049,A -85,B 0,C 180,E1 17064.644,E2 17064.644} C_VEL
LIN {X 0,Y 366.083,Z 402.69,A -85,B 0,C 180,E1 17063.991,E2 17063.991} C_VEL
LIN {X 0,Y 369.077,Z 397.118,A -85,B 0,C 180,E1 17063.512,E2 17063.512} C_VEL
LIN {X 0,Y 372.359,Z 394.885,A -85,B 0,C 180,E1 17062.878,E2 17062.878} C_VEL
LIN {X 0,Y 376.321,Z 389.945,A -85,B 0,C 180,E1 17062.21,E2 17062.21} C_VEL
LIN {X 0,Y 379.783,Z 384.421,A -85,B 0,C 180,E1 17061.683,E2 17061.683} C_VEL
LIN {X 0,Y 384.367,Z 381.167,A -85,B 0,C 180,E1 17060.889,E2 17060.889} C_VEL
LIN {X 0,Y 398.515,Z 373.333,A -85,B 0,C 180,E1 17058.573,E2 17058.573} C_VEL
